KUKA KRL program: EPS_2_251349_MH91A_A_20250929014705.src

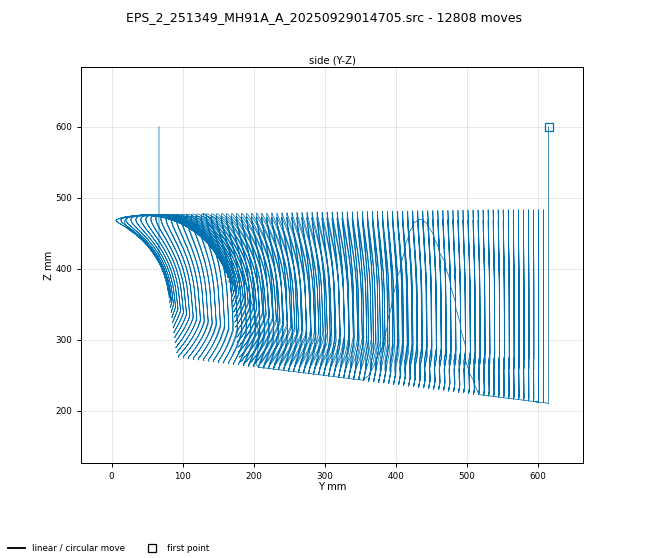
[picture p0: tool path of EPS_2_251349_MH91A_A_20250929014705.src, 12808 of 12810 moves have a stored position in this frame; points joined in program order, loops and branches not executed]
&ACCESS RVP
&REL 4
&COMMENT QRS 19112012
&PARAM EDITMASK = *
DEF PART()
EXT BAS (BAS_COMMAND :IN,REAL :IN )
INT I
BAS (#INITMOV,0 )

;KUKA QRS Post kuka4.cps  Date:22-06-2017 !

File_ID=2865

QRS_PRE_INIT()

;Init var - Until changes are made in qrs_pre_init
Outlet_Square_prg=0
Inlet_1_Square_prg=0
Inlet_2_Square_prg=0
Inlet_3_Square_prg=0
Inlet_4_Square_prg=0
Inlet_5_Square_prg=0

Outlet_1={X 0.000, Y 540.910, Z 382.500, B 0.000, E1 0.000 }
Inlet_1={X 0.000, Y 541.980, Z 367.500, B 0.000, E1 162.000 }
Outlet_1_type=201
Inlet_1_type=201
;QRS#1=Sidecore dimensions
;QRS#2=200-8" PVC SDR 35
;QRS#3=200-8" PVC SDR 35
;QRS#4=
;QRS#5=
;QRS#6=
;QRS#7=
;QRS#8=
;QRS#9=12-08 PSX
;QRS#10=12-08 PSX
;QRS#11=
;QRS#12=
;QRS#13=
;QRS#14=
;QRS#15=
;QRS#16=1220x127x762 2,5'
;QRS#17=EPS Height
;QRS#18=483
;QRS#19=*
;QRS#20= UPDATED VERSION 22-06-2017
;QRS#21=*
Outlet_Square=0100
Inlet_1_Square=0100
Inlet_2_Square=0
Inlet_3_Square=0
Inlet_4_Square=0
Inlet_5_Square=0
Mill_Square=1
Outlet_Square_Prg=204
Inlet_1_Square_prg=204

QRS_INIT()

$ADVANCE=5

; T1
PTP {E1 173.625,E2 173.625}
PTP {X 0,Y 615.486,A -85,B 0,C 180,E1 173.625,E2 173.625,E3 0,E4 0,E5 0,E6 0}
QRS_SPEED_INIT()
LIN {X 0,Y 615.486,Z 600,A -85,B 0,C 180,E1 173.625,E2 173.625,E3 0,E4 0,E5 0,E6 0} C_VEL
LIN {X 0,Y 615.486,Z 220.377,A -85,B 0,C 180,E1 173.625,E2 173.625} C_VEL
LIN {X 0,Y 615.486,Z 212.197,A -85,B 0,C 180,E1 173.625,E2 173.625} C_VEL
LIN {X 0,Y 615.466,Z 210.197,A -85,B 0,C 180,E1 173.439,E2 173.439} C_VEL
LIN {X 0,Y 615.443,Z 210.191,A -85,B 0,C 180,E1 170.804,E2 170.804} C_VEL
LIN {X 0,Y 615.481,Z 210.185,A -85,B 0,C 180,E1 168.143,E2 168.143} C_VEL
LIN {X 0,Y 615.489,Z 210.202,A -85,B 0,C 180,E1 165.455,E2 165.455} C_VEL
LIN {X 0,Y 615.443,Z 210.194,A -85,B 0,C 180,E1 162.732,E2 162.732} C_VEL
LIN {X 0,Y 615.445,Z 210.194,A -85,B 0,C 180,E1 160.665,E2 160.665} C_VEL
LIN {X 0,Y 615.444,Z 210.193,A -85,B 0,C 180,E1 158.571,E2 158.571} C_VEL
LIN {X 0,Y 615.452,Z 210.188,A -85,B 0,C 180,E1 155.999,E2 155.999} C_VEL
LIN {X 0,Y 615.482,Z 210.186,A -85,B 0,C 180,E1 153.56,E2 153.56} C_VEL
LIN {X 0,Y 615.461,Z 210.197,A -85,B 0,C 180,E1 150.597,E2 150.597} C_VEL
LIN {X 0,Y 615.446,Z 210.195,A -85,B 0,C 180,E1 148.317,E2 148.317} C_VEL
LIN {X 0,Y 615.438,Z 210.193,A -85,B 0,C 180,E1 145.98,E2 145.98} C_VEL
LIN {X 0,Y 615.487,Z 210.188,A -85,B 0,C 180,E1 143.064,E2 143.064} C_VEL
LIN {X 0,Y 615.463,Z 210.197,A -85,B 0,C 180,E1 140.254,E2 140.254} C_VEL
LIN {X 0,Y 615.436,Z 210.193,A -85,B 0,C 180,E1 137.649,E2 137.649} C_VEL
LIN {X 0,Y 615.459,Z 210.188,A -85,B 0,C 180,E1 135.071,E2 135.071} C_VEL
LIN {X 0,Y 615.476,Z 210.199,A -85,B 0,C 180,E1 132.086,E2 132.086} C_VEL
LIN {X 0,Y 615.45,Z 210.197,A -85,B 0,C 180,E1 129.753,E2 129.753} C_VEL
LIN {X 0,Y 615.496,Z 210.293,A -85,B 0,C 180,E1 128.068,E2 128.068} C_VEL
LIN {X 0,Y 615.498,Z 215.243,A -85,B 0,C 180,E1 127.241,E2 127.241} C_VEL
LIN {X 0,Y 615.482,Z 234.736,A -85,B 0,C 180,E1 124.194,E2 124.194} C_VEL
LIN {X 0,Y 615.483,Z 252.922,A -85,B 0,C 180,E1 121.388,E2 121.388} C_VEL
LIN {X 0,Y 615.458,Z 256.698,A -85,B 0,C 180,E1 120.85,E2 120.85} C_VEL
LIN {X 0,Y 615.458,Z 257.958,A -85,B 0,C 180,E1 120.802,E2 120.802} C_VEL
LIN {X 0,Y 615.498,Z 364.551,A -85,B 0,C 180,E1 119.531,E2 119.531} C_VEL
LIN {X 0,Y 615.497,Z 378.331,A -85,B 0,C 180,E1 119.218,E2 119.218} C_VEL
LIN {X 0,Y 615.497,Z 390.792,A -85,B 0,C 180,E1 118.798,E2 118.798} C_VEL
LIN {X 0,Y 615.495,Z 402.578,A -85,B 0,C 180,E1 118.257,E2 118.257} C_VEL
LIN {X 0,Y 615.491,Z 414.616,A -85,B 0,C 180,E1 117.545,E2 117.545} C_VEL
LIN {X 0,Y 615.499,Z 425.233,A -85,B 0,C 180,E1 116.751,E2 116.751} C_VEL
LIN {X 0,Y 615.497,Z 434.39,A -85,B 0,C 180,E1 115.897,E2 115.897} C_VEL
LIN {X 0,Y 615.497,Z 442.433,A -85,B 0,C 180,E1 114.991,E2 114.991} C_VEL
LIN {X 0,Y 615.495,Z 449.385,A -85,B 0,C 180,E1 114.023,E2 114.023} C_VEL
LIN {X 0,Y 615.495,Z 454.185,A -85,B 0,C 180,E1 113.2,E2 113.2} C_VEL
LIN {X 0,Y 615.498,Z 459.174,A -85,B 0,C 180,E1 112.136,E2 112.136} C_VEL
LIN {X 0,Y 615.495,Z 462.866,A -85,B 0,C 180,E1 111.081,E2 111.081} C_VEL
LIN {X 0,Y 615.495,Z 465.411,A -85,B 0,C 180,E1 110.033,E2 110.033} C_VEL
LIN {X 0,Y 615.496,Z 466.492,A -85,B 0,C 180,E1 109.338,E2 109.338} C_VEL
LIN {X 0,Y 615.494,Z 467.164,A -85,B 0,C 180,E1 108.624,E2 108.624} C_VEL
LIN {X 0,Y 615.498,Z 467.388,A -85,B 0,C 180,E1 107.957,E2 107.957} C_VEL
LIN {X 0,Y 615.494,Z 467.152,A -85,B 0,C 180,E1 107.27,E2 107.27} C_VEL
LIN {X 0,Y 615.496,Z 466.353,A -85,B 0,C 180,E1 106.453,E2 106.453} C_VEL
LIN {X 0,Y 615.496,Z 463.937,A -85,B 0,C 180,E1 105.226,E2 105.226} C_VEL
LIN {X 0,Y 615.496,Z 459.888,A -85,B 0,C 180,E1 103.959,E2 103.959} C_VEL
LIN {X 0,Y 615.496,Z 455.011,A -85,B 0,C 180,E1 102.865,E2 102.865} C_VEL
LIN {X 0,Y 615.5,Z 448.085,A -85,B 0,C 180,E1 101.694,E2 101.694} C_VEL
LIN {X 0,Y 615.498,Z 440.842,A -85,B 0,C 180,E1 100.724,E2 100.724} C_VEL
LIN {X 0,Y 615.497,Z 434.547,A -85,B 0,C 180,E1 100.028,E2 100.028} C_VEL
LIN {X 0,Y 615.499,Z 425.695,A -85,B 0,C 180,E1 99.199,E2 99.199} C_VEL
LIN {X 0,Y 615.487,Z 415.964,A -85,B 0,C 180,E1 98.454,E2 98.454} C_VEL
LIN {X 0,Y 615.471,Z 405.228,A -85,B 0,C 180,E1 97.793,E2 97.793} C_VEL
LIN {X 0,Y 615.497,Z 393.247,A -85,B 0,C 180,E1 97.216,E2 97.216} C_VEL
LIN {X 0,Y 615.499,Z 381.306,A -85,B 0,C 180,E1 96.78,E2 96.78} C_VEL
LIN {X 0,Y 615.498,Z 368.629,A -85,B 0,C 180,E1 96.454,E2 96.454} C_VEL
LIN {X 0,Y 615.499,Z 353.252,A -85,B 0,C 180,E1 96.228,E2 96.228} C_VEL
LIN {X 0,Y 615.488,Z 257.435,A -85,B 0,C 180,E1 95.098,E2 95.098} C_VEL
LIN {X 0,Y 615.488,Z 256.065,A -85,B 0,C 180,E1 94.995,E2 94.995} C_VEL
LIN {X 0,Y 615.46,Z 238.445,A -85,B 0,C 180,E1 92.291,E2 92.291} C_VEL
LIN {X 0,Y 615.429,Z 222.697,A -85,B 0,C 180,E1 89.837,E2 89.837} C_VEL
LIN {X 0,Y 615.494,Z 210.317,A -85,B 0,C 180,E1 87.853,E2 87.853} C_VEL
LIN {X 0,Y 615.483,Z 210.193,A -85,B 0,C 180,E1 85.416,E2 85.416} C_VEL
LIN {X 0,Y 615.486,Z 210.181,A -85,B 0,C 180,E1 82.785,E2 82.785} C_VEL
LIN {X 0,Y 615.469,Z 210.187,A -85,B 0,C 180,E1 80.138,E2 80.138} C_VEL
LIN {X 0,Y 615.492,Z 210.199,A -85,B 0,C 180,E1 77.47,E2 77.47} C_VEL
LIN {X 0,Y 615.481,Z 210.187,A -85,B 0,C 180,E1 74.774,E2 74.774} C_VEL
LIN {X 0,Y 615.477,Z 210.183,A -85,B 0,C 180,E1 72.043,E2 72.043} C_VEL
LIN {X 0,Y 615.481,Z 210.196,A -85,B 0,C 180,E1 69.269,E2 69.269} C_VEL
LIN {X 0,Y 615.482,Z 210.187,A -85,B 0,C 180,E1 66.444,E2 66.444} C_VEL
LIN {X 0,Y 615.479,Z 210.186,A -85,B 0,C 180,E1 64.284,E2 64.284} C_VEL
LIN {X 0,Y 615.471,Z 210.185,A -85,B 0,C 180,E1 61.541,E2 61.541} C_VEL
LIN {X 0,Y 615.477,Z 210.195,A -85,B 0,C 180,E1 58.906,E2 58.906} C_VEL
LIN {X 0,Y 615.492,Z 210.197,A -85,B 0,C 180,E1 56.456,E2 56.456} C_VEL
LIN {X 0,Y 615.483,Z 210.181,A -85,B 0,C 180,E1 53.575,E2 53.575} C_VEL
LIN {X 0,Y 615.467,Z 210.188,A -85,B 0,C 180,E1 50.932,E2 50.932} C_VEL
LIN {X 0,Y 615.476,Z 210.195,A -85,B 0,C 180,E1 48.526,E2 48.526} C_VEL
LIN {X 0,Y 615.484,Z 210.193,A -85,B 0,C 180,E1 45.851,E2 45.851} C_VEL
LIN {X 0,Y 615.483,Z 210.181,A -85,B 0,C 180,E1 43.048,E2 43.048} C_VEL
LIN {X 0,Y 615.468,Z 210.187,A -85,B 0,C 180,E1 40.602,E2 40.602} C_VEL
LIN {X 0,Y 615.477,Z 210.198,A -85,B 0,C 180,E1 38.011,E2 38.011} C_VEL
LIN {X 0,Y 615.491,Z 210.197,A -85,B 0,C 180,E1 35.61,E2 35.61} C_VEL
LIN {X 0,Y 615.482,Z 210.189,A -85,B 0,C 180,E1 33.231,E2 33.231} C_VEL
LIN {X 0,Y 615.484,Z 210.184,A -85,B 0,C 180,E1 30.915,E2 30.915} C_VEL
LIN {X 0,Y 615.482,Z 210.181,A -85,B 0,C 180,E1 28.45,E2 28.45} C_VEL
LIN {X 0,Y 615.478,Z 210.196,A -85,B 0,C 180,E1 25.568,E2 25.568} C_VEL
LIN {X 0,Y 615.482,Z 210.19,A -85,B 0,C 180,E1 22.84,E2 22.84} C_VEL
LIN {X 0,Y 615.477,Z 210.182,A -85,B 0,C 180,E1 20.029,E2 20.029} C_VEL
LIN {X 0,Y 615.473,Z 210.196,A -85,B 0,C 180,E1 17.267,E2 17.267} C_VEL
LIN {X 0,Y 615.483,Z 210.191,A -85,B 0,C 180,E1 14.545,E2 14.545} C_VEL
LIN {X 0,Y 615.485,Z 210.181,A -85,B 0,C 180,E1 11.857,E2 11.857} C_VEL
LIN {X 0,Y 615.466,Z 210.191,A -85,B 0,C 180,E1 9.196,E2 9.196} C_VEL
LIN {X 0,Y 615.489,Z 210.201,A -85,B 0,C 180,E1 6.553,E2 6.553} C_VEL
LIN {X 0,Y 615.485,Z 210.185,A -85,B 0,C 180,E1 3.925,E2 3.925} C_VEL
LIN {X 0,Y 615.477,Z 210.182,A -85,B 0,C 180,E1 1.306,E2 1.306} C_VEL
LIN {X 0,Y 615.468,Z 210.192,A -85,B 0,C 180,E1 -1.312,E2 -1.312} C_VEL
LIN {X 0,Y 615.488,Z 210.199,A -85,B 0,C 180,E1 -3.931,E2 -3.931} C_VEL
LIN {X 0,Y 615.484,Z 210.184,A -85,B 0,C 180,E1 -6.58,E2 -6.58} C_VEL
LIN {X 0,Y 615.471,Z 210.184,A -85,B 0,C 180,E1 -9.202,E2 -9.202} C_VEL
LIN {X 0,Y 615.474,Z 210.195,A -85,B 0,C 180,E1 -11.863,E2 -11.863} C_VEL
LIN {X 0,Y 615.484,Z 210.192,A -85,B 0,C 180,E1 -14.551,E2 -14.551} C_VEL
LIN {X 0,Y 615.487,Z 210.18,A -85,B 0,C 180,E1 -17.273,E2 -17.273} C_VEL
LIN {X 0,Y 615.465,Z 210.192,A -85,B 0,C 180,E1 -20.036,E2 -20.036} C_VEL
LIN {X 0,Y 615.486,Z 210.193,A -85,B 0,C 180,E1 -22.847,E2 -22.847} C_VEL
LIN {X 0,Y 615.479,Z 210.182,A -85,B 0,C 180,E1 -25.718,E2 -25.718} C_VEL
LIN {X 0,Y 615.47,Z 210.194,A -85,B 0,C 180,E1 -28.448,E2 -28.448} C_VEL
LIN {X 0,Y 615.483,Z 210.197,A -85,B 0,C 180,E1 -31.086,E2 -31.086} C_VEL
LIN {X 0,Y 615.478,Z 210.182,A -85,B 0,C 180,E1 -34.024,E2 -34.024} C_VEL
LIN {X 0,Y 615.463,Z 210.188,A -85,B 0,C 180,E1 -36.428,E2 -36.428} C_VEL
LIN {X 0,Y 615.483,Z 210.197,A -85,B 0,C 180,E1 -39.062,E2 -39.062} C_VEL
LIN {X 0,Y 615.49,Z 210.196,A -85,B 0,C 180,E1 -41.475,E2 -41.475} C_VEL
LIN {X 0,Y 615.495,Z 210.18,A -85,B 0,C 180,E1 -44.15,E2 -44.15} C_VEL
LIN {X 0,Y 615.463,Z 210.19,A -85,B 0,C 180,E1 -46.956,E2 -46.956} C_VEL
LIN {X 0,Y 615.477,Z 210.196,A -85,B 0,C 180,E1 -49.393,E2 -49.393} C_VEL
LIN {X 0,Y 615.486,Z 210.193,A -85,B 0,C 180,E1 -51.99,E2 -51.99} C_VEL
LIN {X 0,Y 615.487,Z 210.185,A -85,B 0,C 180,E1 -54.385,E2 -54.385} C_VEL
LIN {X 0,Y 615.487,Z 210.181,A -85,B 0,C 180,E1 -56.764,E2 -56.764} C_VEL
LIN {X 0,Y 615.474,Z 210.183,A -85,B 0,C 180,E1 -59.08,E2 -59.08} C_VEL
LIN {X 0,Y 615.463,Z 210.19,A -85,B 0,C 180,E1 -61.555,E2 -61.555} C_VEL
LIN {X 0,Y 615.496,Z 210.198,A -85,B 0,C 180,E1 -64.285,E2 -64.285} C_VEL
LIN {X 0,Y 615.484,Z 210.181,A -85,B 0,C 180,E1 -67.156,E2 -67.156} C_VEL
LIN {X 0,Y 615.492,Z 210.44,A -85,B 0,C 180,E1 -68.481,E2 -68.481} C_VEL
LIN {X 0,Y 615.494,Z 228.962,A -85,B 0,C 180,E1 -71.182,E2 -71.182} C_VEL
LIN {X 0,Y 615.488,Z 249.426,A -85,B 0,C 180,E1 -74.095,E2 -74.095} C_VEL
LIN {X 0,Y 615.473,Z 268.666,A -85,B 0,C 180,E1 -76.799,E2 -76.799} C_VEL
LIN {X 0,Y 615.487,Z 271.254,A -85,B 0,C 180,E1 -77.114,E2 -77.114} C_VEL
LIN {X 0,Y 615.491,Z 280.067,A -85,B 0,C 180,E1 -77.24,E2 -77.24} C_VEL
LIN {X 0,Y 615.498,Z 378.843,A -85,B 0,C 180,E1 -78.411,E2 -78.411} C_VEL
LIN {X 0,Y 615.498,Z 391.352,A -85,B 0,C 180,E1 -78.682,E2 -78.682} C_VEL
LIN {X 0,Y 615.496,Z 404.516,A -85,B 0,C 180,E1 -79.109,E2 -79.109} C_VEL
LIN {X 0,Y 615.491,Z 416.482,A -85,B 0,C 180,E1 -79.64,E2 -79.64} C_VEL
LIN {X 0,Y 615.48,Z 428,A -85,B 0,C 180,E1 -80.304,E2 -80.304} C_VEL
LIN {X 0,Y 615.499,Z 438.344,A -85,B 0,C 180,E1 -81.05,E2 -81.05} C_VEL
LIN {X 0,Y 615.498,Z 446.694,A -85,B 0,C 180,E1 -81.794,E2 -81.794} C_VEL
LIN {X 0,Y 615.498,Z 454.608,A -85,B 0,C 180,E1 -82.62,E2 -82.62} C_VEL
LIN {X 0,Y 615.49,Z 462.206,A -85,B 0,C 180,E1 -83.608,E2 -83.608} C_VEL
LIN {X 0,Y 615.498,Z 469.206,A -85,B 0,C 180,E1 -84.759,E2 -84.759} C_VEL
LIN {X 0,Y 615.493,Z 473.852,A -85,B 0,C 180,E1 -85.744,E2 -85.744} C_VEL
LIN {X 0,Y 615.494,Z 477.399,A -85,B 0,C 180,E1 -86.727,E2 -86.727} C_VEL
LIN {X 0,Y 615.497,Z 479.233,A -85,B 0,C 180,E1 -87.382,E2 -87.382} C_VEL
LIN {X 0,Y 615.497,Z 480.609,A -85,B 0,C 180,E1 -88.037,E2 -88.037} C_VEL
LIN {X 0,Y 615.496,Z 482.174,A -85,B 0,C 180,E1 -89.346,E2 -89.346} C_VEL
LIN {X 0,Y 615.494,Z 482.389,A -85,B 0,C 180,E1 -90,E2 -90} C_VEL
LIN {X 0,Y 615.495,Z 481.58,A -85,B 0,C 180,E1 -91.309,E2 -91.309} C_VEL
LIN {X 0,Y 615.497,Z 480.608,A -85,B 0,C 180,E1 -91.963,E2 -91.963} C_VEL
LIN {X 0,Y 615.497,Z 479.232,A -85,B 0,C 180,E1 -92.618,E2 -92.618} C_VEL
LIN {X 0,Y 615.496,Z 476.349,A -85,B 0,C 180,E1 -93.601,E2 -93.601} C_VEL
LIN {X 0,Y 615.498,Z 472.441,A -85,B 0,C 180,E1 -94.585,E2 -94.585} C_VEL
LIN {X 0,Y 615.499,Z 467.404,A -85,B 0,C 180,E1 -95.57,E2 -95.57} C_VEL
LIN {X 0,Y 615.489,Z 460.919,A -85,B 0,C 180,E1 -96.577,E2 -96.577} C_VEL
LIN {X 0,Y 615.497,Z 453.131,A -85,B 0,C 180,E1 -97.546,E2 -97.546} C_VEL
LIN {X 0,Y 615.498,Z 443.255,A -85,B 0,C 180,E1 -98.537,E2 -98.537} C_VEL
LIN {X 0,Y 615.495,Z 432.863,A -85,B 0,C 180,E1 -99.365,E2 -99.365} C_VEL
LIN {X 0,Y 615.475,Z 422.574,A -85,B 0,C 180,E1 -100.029,E2 -100.029} C_VEL
LIN {X 0,Y 615.497,Z 411.095,A -85,B 0,C 180,E1 -100.618,E2 -100.618} C_VEL
LIN {X 0,Y 615.499,Z 399.268,A -85,B 0,C 180,E1 -101.08,E2 -101.08} C_VEL
LIN {X 0,Y 615.498,Z 386.231,A -85,B 0,C 180,E1 -101.443,E2 -101.443} C_VEL
LIN {X 0,Y 615.499,Z 372.923,A -85,B 0,C 180,E1 -101.673,E2 -101.673} C_VEL
LIN {X 0,Y 615.487,Z 271.727,A -85,B 0,C 180,E1 -102.866,E2 -102.866} C_VEL
LIN {X 0,Y 615.485,Z 270.517,A -85,B 0,C 180,E1 -102.95,E2 -102.95} C_VEL
LIN {X 0,Y 615.482,Z 250.626,A -85,B 0,C 180,E1 -105.735,E2 -105.735} C_VEL
LIN {X 0,Y 615.491,Z 231.585,A -85,B 0,C 180,E1 -108.443,E2 -108.443} C_VEL
LIN {X 0,Y 615.492,Z 212.09,A -85,B 0,C 180,E1 -111.256,E2 -111.256} C_VEL
LIN {X 0,Y 615.49,Z 210.313,A -85,B 0,C 180,E1 -111.564,E2 -111.564} C_VEL
LIN {X 0,Y 615.462,Z 210.19,A -85,B 0,C 180,E1 -114.273,E2 -114.273} C_VEL
LIN {X 0,Y 615.497,Z 210.179,A -85,B 0,C 180,E1 -117.045,E2 -117.045} C_VEL
LIN {X 0,Y 615.493,Z 210.197,A -85,B 0,C 180,E1 -119.794,E2 -119.794} C_VEL
LIN {X 0,Y 615.463,Z 210.192,A -85,B 0,C 180,E1 -122.459,E2 -122.459} C_VEL
LIN {X 0,Y 615.46,Z 210.188,A -85,B 0,C 180,E1 -124.817,E2 -124.817} C_VEL
LIN {X 0,Y 615.478,Z 210.182,A -85,B 0,C 180,E1 -127.243,E2 -127.243} C_VEL
LIN {X 0,Y 615.49,Z 210.195,A -85,B 0,C 180,E1 -130.088,E2 -130.088} C_VEL
LIN {X 0,Y 615.499,Z 210.2,A -85,B 0,C 180,E1 -132.352,E2 -132.352} C_VEL
LIN {X 0,Y 615.455,Z 210.191,A -85,B 0,C 180,E1 -135.072,E2 -135.072} C_VEL
LIN {X 0,Y 615.497,Z 210.181,A -85,B 0,C 180,E1 -137.919,E2 -137.919} C_VEL
LIN {X 0,Y 615.487,Z 210.189,A -85,B 0,C 180,E1 -140.248,E2 -140.248} C_VEL
LIN {X 0,Y 615.467,Z 210.195,A -85,B 0,C 180,E1 -143.066,E2 -143.066} C_VEL
LIN {X 0,Y 615.458,Z 210.193,A -85,B 0,C 180,E1 -145.303,E2 -145.303} C_VEL
LIN {X 0,Y 615.456,Z 210.189,A -85,B 0,C 180,E1 -147.674,E2 -147.674} C_VEL
LIN {X 0,Y 615.482,Z 210.183,A -85,B 0,C 180,E1 -150.206,E2 -150.206} C_VEL
LIN {X 0,Y 615.493,Z 210.196,A -85,B 0,C 180,E1 -152.954,E2 -152.954} C_VEL
LIN {X 0,Y 615.452,Z 210.193,A -85,B 0,C 180,E1 -155.724,E2 -155.724} C_VEL
LIN {X 0,Y 615.453,Z 210.192,A -85,B 0,C 180,E1 -157.86,E2 -157.86} C_VEL
LIN {X 0,Y 615.45,Z 210.192,A -85,B 0,C 180,E1 -159.964,E2 -159.964} C_VEL
LIN {X 0,Y 615.452,Z 210.191,A -85,B 0,C 180,E1 -162.04,E2 -162.04} C_VEL
LIN {X 0,Y 615.483,Z 210.183,A -85,B 0,C 180,E1 -164.772,E2 -164.772} C_VEL
LIN {X 0,Y 615.489,Z 210.197,A -85,B 0,C 180,E1 -167.467,E2 -167.467} C_VEL
LIN {X 0,Y 615.457,Z 210.194,A -85,B 0,C 180,E1 -170.135,E2 -170.135} C_VEL
LIN {X 0,Y 615.457,Z 210.187,A -85,B 0,C 180,E1 -172.781,E2 -172.781} C_VEL
LIN {X 0,Y 615.495,Z 210.185,A -85,B 0,C 180,E1 -175.413,E2 -175.413} C_VEL
LIN {X 0,Y 615.492,Z 210.199,A -85,B 0,C 180,E1 -178.034,E2 -178.034} C_VEL
LIN {X 0,Y 615.449,Z 210.193,A -85,B 0,C 180,E1 -180.651,E2 -180.651} C_VEL
LIN {X 0,Y 615.46,Z 210.187,A -85,B 0,C 180,E1 -183.27,E2 -183.27} C_VEL
LIN {X 0,Y 615.494,Z 210.188,A -85,B 0,C 180,E1 -185.895,E2 -185.895} C_VEL
LIN {X 0,Y 615.466,Z 210.197,A -85,B 0,C 180,E1 -186.561,E2 -186.561} C_VEL
LIN {X 0,Y 614.775,Z 210.337,A -85,B 0,C 180,E1 -187.107,E2 -187.107} C_VEL
LIN {X 0,Y 611.924,Z 210.759,A -85,B 0,C 180,E1 -187.993,E2 -187.993} C_VEL
LIN {X 0,Y 609.535,Z 211.065,A -85,B 0,C 180,E1 -188.706,E2 -188.706} C_VEL
LIN {X 0,Y 608.516,Z 211.18,A -85,B 0,C 180,E1 -189.256,E2 -189.256} C_VEL
LIN {X 0,Y 608.436,Z 211.188,A -85,B 0,C 180,E1 -189.442,E2 -189.442} C_VEL
LIN {X 0,Y 608.458,Z 211.189,A -85,B 0,C 180,E1 -191.996,E2 -191.996} C_VEL
LIN {X 0,Y 608.466,Z 211.193,A -85,B 0,C 180,E1 -194.717,E2 -194.717} C_VEL
LIN {X 0,Y 608.419,Z 211.191,A -85,B 0,C 180,E1 -197.474,E2 -197.474} C_VEL
LIN {X 0,Y 608.421,Z 211.19,A -85,B 0,C 180,E1 -199.568,E2 -199.568} C_VEL
LIN {X 0,Y 608.436,Z 211.188,A -85,B 0,C 180,E1 -201.688,E2 -201.688} C_VEL
LIN {X 0,Y 608.447,Z 211.192,A -85,B 0,C 180,E1 -204.567,E2 -204.567} C_VEL
LIN {X 0,Y 608.425,Z 211.193,A -85,B 0,C 180,E1 -207.514,E2 -207.514} C_VEL
LIN {X 0,Y 608.426,Z 211.19,A -85,B 0,C 180,E1 -209.965,E2 -209.965} C_VEL
LIN {X 0,Y 608.437,Z 211.189,A -85,B 0,C 180,E1 -212.519,E2 -212.519} C_VEL
LIN {X 0,Y 608.432,Z 211.2,A -85,B 0,C 180,E1 -215.273,E2 -215.273} C_VEL
LIN {X 0,Y 608.441,Z 211.193,A -85,B 0,C 180,E1 -217.743,E2 -217.743} C_VEL
LIN {X 0,Y 608.409,Z 211.192,A -85,B 0,C 180,E1 -220.324,E2 -220.324} C_VEL
LIN {X 0,Y 608.436,Z 211.19,A -85,B 0,C 180,E1 -222.955,E2 -222.955} C_VEL
LIN {X 0,Y 608.441,Z 211.199,A -85,B 0,C 180,E1 -225.731,E2 -225.731} C_VEL
LIN {X 0,Y 608.453,Z 211.194,A -85,B 0,C 180,E1 -227.938,E2 -227.938} C_VEL
LIN {X 0,Y 608.433,Z 211.19,A -85,B 0,C 180,E1 -230.699,E2 -230.699} C_VEL
LIN {X 0,Y 608.503,Z 211.414,A -85,B 0,C 180,E1 -231.896,E2 -231.896} C_VEL
LIN {X 0,Y 608.479,Z 227.922,A -85,B 0,C 180,E1 -234.529,E2 -234.529} C_VEL
LIN {X 0,Y 608.48,Z 244.489,A -85,B 0,C 180,E1 -237.122,E2 -237.122} C_VEL
LIN {X 0,Y 608.457,Z 256.895,A -85,B 0,C 180,E1 -239.009,E2 -239.009} C_VEL
LIN {X 0,Y 608.559,Z 259.904,A -85,B 0,C 180,E1 -239.075,E2 -239.075} C_VEL
LIN {X 0,Y 608.55,Z 364.504,A -85,B 0,C 180,E1 -240.332,E2 -240.332} C_VEL
LIN {X 0,Y 608.543,Z 377.632,A -85,B 0,C 180,E1 -240.629,E2 -240.629} C_VEL
LIN {X 0,Y 608.532,Z 389.978,A -85,B 0,C 180,E1 -241.041,E2 -241.041} C_VEL
LIN {X 0,Y 608.511,Z 402.259,A -85,B 0,C 180,E1 -241.598,E2 -241.598} C_VEL
LIN {X 0,Y 608.498,Z 414.13,A -85,B 0,C 180,E1 -242.298,E2 -242.298} C_VEL
LIN {X 0,Y 608.487,Z 424.611,A -85,B 0,C 180,E1 -243.072,E2 -243.072} C_VEL
LIN {X 0,Y 608.458,Z 434.253,A -85,B 0,C 180,E1 -243.965,E2 -243.965} C_VEL
LIN {X 0,Y 608.455,Z 442.443,A -85,B 0,C 180,E1 -244.882,E2 -244.882} C_VEL
LIN {X 0,Y 608.454,Z 449.372,A -85,B 0,C 180,E1 -245.839,E2 -245.839} C_VEL
LIN {X 0,Y 608.436,Z 455.39,A -85,B 0,C 180,E1 -246.875,E2 -246.875} C_VEL
LIN {X 0,Y 608.452,Z 460.23,A -85,B 0,C 180,E1 -247.951,E2 -247.951} C_VEL
LIN {X 0,Y 608.438,Z 463.798,A -85,B 0,C 180,E1 -249.018,E2 -249.018} C_VEL
LIN {X 0,Y 608.434,Z 465.533,A -85,B 0,C 180,E1 -249.725,E2 -249.725} C_VEL
LIN {X 0,Y 608.436,Z 466.815,A -85,B 0,C 180,E1 -250.429,E2 -250.429} C_VEL
LIN {X 0,Y 608.437,Z 467.708,A -85,B 0,C 180,E1 -251.276,E2 -251.276} C_VEL
LIN {X 0,Y 608.437,Z 467.894,A -85,B 0,C 180,E1 -252.523,E2 -252.523} C_VEL
LIN {X 0,Y 608.424,Z 467.07,A -85,B 0,C 180,E1 -253.466,E2 -253.466} C_VEL
LIN {X 0,Y 608.42,Z 465.042,A -85,B 0,C 180,E1 -254.593,E2 -254.593} C_VEL
LIN {X 0,Y 608.441,Z 462.112,A -85,B 0,C 180,E1 -255.62,E2 -255.62} C_VEL
LIN {X 0,Y 608.442,Z 458.121,A -85,B 0,C 180,E1 -256.643,E2 -256.643} C_VEL
LIN {X 0,Y 608.437,Z 451.97,A -85,B 0,C 180,E1 -257.83,E2 -257.83} C_VEL
LIN {X 0,Y 608.445,Z 444.669,A -85,B 0,C 180,E1 -258.921,E2 -258.921} C_VEL
LIN {X 0,Y 608.477,Z 436.901,A -85,B 0,C 180,E1 -259.855,E2 -259.855} C_VEL
LIN {X 0,Y 608.467,Z 426.444,A -85,B 0,C 180,E1 -260.862,E2 -260.862} C_VEL
LIN {X 0,Y 608.471,Z 415.564,A -85,B 0,C 180,E1 -261.699,E2 -261.699} C_VEL
LIN {X 0,Y 608.492,Z 404.602,A -85,B 0,C 180,E1 -262.367,E2 -262.367} C_VEL
LIN {X 0,Y 608.542,Z 391.798,A -85,B 0,C 180,E1 -262.976,E2 -262.976} C_VEL
LIN {X 0,Y 608.532,Z 379.509,A -85,B 0,C 180,E1 -263.41,E2 -263.41} C_VEL
LIN {X 0,Y 608.565,Z 366.436,A -85,B 0,C 180,E1 -263.722,E2 -263.722} C_VEL
LIN {X 0,Y 608.55,Z 346.3,A -85,B 0,C 180,E1 -263.992,E2 -263.992} C_VEL
LIN {X 0,Y 608.537,Z 257.452,A -85,B 0,C 180,E1 -265.052,E2 -265.052} C_VEL
LIN {X 0,Y 608.463,Z 256.535,A -85,B 0,C 180,E1 -265.113,E2 -265.113} C_VEL
LIN {X 0,Y 608.458,Z 238.843,A -85,B 0,C 180,E1 -267.848,E2 -267.848} C_VEL
LIN {X 0,Y 608.447,Z 223.051,A -85,B 0,C 180,E1 -270.331,E2 -270.331} C_VEL
LIN {X 0,Y 608.5,Z 211.284,A -85,B 0,C 180,E1 -272.234,E2 -272.234} C_VEL
LIN {X 0,Y 608.485,Z 211.182,A -85,B 0,C 180,E1 -275.301,E2 -275.301} C_VEL
LIN {X 0,Y 608.456,Z 211.189,A -85,B 0,C 180,E1 -277.967,E2 -277.967} C_VEL
LIN {X 0,Y 608.462,Z 211.195,A -85,B 0,C 180,E1 -280.65,E2 -280.65} C_VEL
LIN {X 0,Y 608.454,Z 211.187,A -85,B 0,C 180,E1 -283.356,E2 -283.356} C_VEL
LIN {X 0,Y 608.467,Z 211.186,A -85,B 0,C 180,E1 -286.093,E2 -286.093} C_VEL
LIN {X 0,Y 608.453,Z 211.198,A -85,B 0,C 180,E1 -288.869,E2 -288.869} C_VEL
LIN {X 0,Y 608.457,Z 211.186,A -85,B 0,C 180,E1 -291.692,E2 -291.692} C_VEL
LIN {X 0,Y 608.44,Z 211.19,A -85,B 0,C 180,E1 -294.571,E2 -294.571} C_VEL
LIN {X 0,Y 608.469,Z 211.195,A -85,B 0,C 180,E1 -297.217,E2 -297.217} C_VEL
LIN {X 0,Y 608.484,Z 211.183,A -85,B 0,C 180,E1 -299.985,E2 -299.985} C_VEL
LIN {X 0,Y 608.447,Z 211.189,A -85,B 0,C 180,E1 -302.88,E2 -302.88} C_VEL
LIN {X 0,Y 608.466,Z 211.192,A -85,B 0,C 180,E1 -305.276,E2 -305.276} C_VEL
LIN {X 0,Y 608.455,Z 211.188,A -85,B 0,C 180,E1 -308.247,E2 -308.247} C_VEL
LIN {X 0,Y 608.472,Z 211.185,A -85,B 0,C 180,E1 -310.339,E2 -310.339} C_VEL
LIN {X 0,Y 608.454,Z 211.189,A -85,B 0,C 180,E1 -313.314,E2 -313.314} C_VEL
LIN {X 0,Y 608.47,Z 211.192,A -85,B 0,C 180,E1 -316.137,E2 -316.137} C_VEL
LIN {X 0,Y 608.455,Z 211.186,A -85,B 0,C 180,E1 -318.83,E2 -318.83} C_VEL
LIN {X 0,Y 608.462,Z 211.185,A -85,B 0,C 180,E1 -321.417,E2 -321.417} C_VEL
LIN {X 0,Y 608.456,Z 211.192,A -85,B 0,C 180,E1 -323.953,E2 -323.953} C_VEL
LIN {X 0,Y 608.461,Z 211.197,A -85,B 0,C 180,E1 -326.334,E2 -326.334} C_VEL
LIN {X 0,Y 608.46,Z 211.191,A -85,B 0,C 180,E1 -328.73,E2 -328.73} C_VEL
LIN {X 0,Y 608.468,Z 211.184,A -85,B 0,C 180,E1 -331.38,E2 -331.38} C_VEL
LIN {X 0,Y 608.436,Z 211.189,A -85,B 0,C 180,E1 -333.969,E2 -333.969} C_VEL
LIN {X 0,Y 608.451,Z 211.188,A -85,B 0,C 180,E1 -336.159,E2 -336.159} C_VEL
LIN {X 0,Y 608.455,Z 211.189,A -85,B 0,C 180,E1 -338.312,E2 -338.312} C_VEL
LIN {X 0,Y 608.446,Z 211.194,A -85,B 0,C 180,E1 -341.134,E2 -341.134} C_VEL
LIN {X 0,Y 608.455,Z 211.185,A -85,B 0,C 180,E1 -343.91,E2 -343.91} C_VEL
LIN {X 0,Y 608.452,Z 211.189,A -85,B 0,C 180,E1 -346.647,E2 -346.647} C_VEL
LIN {X 0,Y 608.464,Z 211.195,A -85,B 0,C 180,E1 -349.354,E2 -349.354} C_VEL
LIN {X 0,Y 608.477,Z 211.184,A -85,B 0,C 180,E1 -352.036,E2 -352.036} C_VEL
LIN {X 0,Y 608.449,Z 211.187,A -85,B 0,C 180,E1 -354.701,E2 -354.701} C_VEL
LIN {X 0,Y 608.472,Z 211.191,A -85,B 0,C 180,E1 -357.355,E2 -357.355} C_VEL
LIN {X 0,Y 608.474,Z 211.189,A -85,B 0,C 180,E1 -360.003,E2 -360.003} C_VEL
LIN {X 0,Y 608.481,Z 211.183,A -85,B 0,C 180,E1 -362.651,E2 -362.651} C_VEL
LIN {X 0,Y 608.448,Z 211.189,A -85,B 0,C 180,E1 -365.305,E2 -365.305} C_VEL
LIN {X 0,Y 608.476,Z 211.195,A -85,B 0,C 180,E1 -367.97,E2 -367.97} C_VEL
LIN {X 0,Y 608.469,Z 211.184,A -85,B 0,C 180,E1 -370.958,E2 -370.958} C_VEL
LIN {X 0,Y 608.456,Z 211.186,A -85,B 0,C 180,E1 -373.359,E2 -373.359} C_VEL
LIN {X 0,Y 608.451,Z 211.194,A -85,B 0,C 180,E1 -376.096,E2 -376.096} C_VEL
LIN {X 0,Y 608.458,Z 211.189,A -85,B 0,C 180,E1 -378.872,E2 -378.872} C_VEL
LIN {X 0,Y 608.463,Z 211.185,A -85,B 0,C 180,E1 -381.694,E2 -381.694} C_VEL
LIN {X 0,Y 608.445,Z 211.198,A -85,B 0,C 180,E1 -384.573,E2 -384.573} C_VEL
LIN {X 0,Y 608.478,Z 211.187,A -85,B 0,C 180,E1 -387.208,E2 -387.208} C_VEL
LIN {X 0,Y 608.443,Z 211.187,A -85,B 0,C 180,E1 -389.968,E2 -389.968} C_VEL
LIN {X 0,Y 608.45,Z 211.196,A -85,B 0,C 180,E1 -392.882,E2 -392.882} C_VEL
LIN {X 0,Y 608.438,Z 211.196,A -85,B 0,C 180,E1 -395.28,E2 -395.28} C_VEL
LIN {X 0,Y 608.47,Z 211.186,A -85,B 0,C 180,E1 -397.748,E2 -397.748} C_VEL
LIN {X 0,Y 608.447,Z 211.187,A -85,B 0,C 180,E1 -400.329,E2 -400.329} C_VEL
LIN {X 0,Y 608.437,Z 211.192,A -85,B 0,C 180,E1 -402.963,E2 -402.963} C_VEL
LIN {X 0,Y 608.453,Z 211.193,A -85,B 0,C 180,E1 -405.738,E2 -405.738} C_VEL
LIN {X 0,Y 608.452,Z 211.186,A -85,B 0,C 180,E1 -408.66,E2 -408.66} C_VEL
LIN {X 0,Y 608.467,Z 211.196,A -85,B 0,C 180,E1 -411.761,E2 -411.761} C_VEL
LIN {X 0,Y 608.436,Z 211.188,A -85,B 0,C 180,E1 -414.722,E2 -414.722} C_VEL
LIN {X 0,Y 608.452,Z 211.187,A -85,B 0,C 180,E1 -417.121,E2 -417.121} C_VEL
LIN {X 0,Y 608.468,Z 211.196,A -85,B 0,C 180,E1 -420.03,E2 -420.03} C_VEL
LIN {X 0,Y 608.486,Z 211.184,A -85,B 0,C 180,E1 -422.793,E2 -422.793} C_VEL
LIN {X 0,Y 608.445,Z 211.188,A -85,B 0,C 180,E1 -425.429,E2 -425.429} C_VEL
LIN {X 0,Y 608.5,Z 211.351,A -85,B 0,C 180,E1 -428.354,E2 -428.354} C_VEL
LIN {X 0,Y 608.545,Z 226.58,A -85,B 0,C 180,E1 -430.608,E2 -430.608} C_VEL
LIN {X 0,Y 608.505,Z 246.378,A -85,B 0,C 180,E1 -433.461,E2 -433.461} C_VEL
LIN {X 0,Y 608.467,Z 266.398,A -85,B 0,C 180,E1 -436.304,E2 -436.304} C_VEL
LIN {X 0,Y 608.497,Z 271.295,A -85,B 0,C 180,E1 -436.963,E2 -436.963} C_VEL
LIN {X 0,Y 608.587,Z 276.532,A -85,B 0,C 180,E1 -437.05,E2 -437.05} C_VEL
LIN {X 0,Y 608.548,Z 378.962,A -85,B 0,C 180,E1 -438.277,E2 -438.277} C_VEL
LIN {X 0,Y 608.548,Z 392.226,A -85,B 0,C 180,E1 -438.572,E2 -438.572} C_VEL
LIN {X 0,Y 608.544,Z 405.347,A -85,B 0,C 180,E1 -439.01,E2 -439.01} C_VEL
LIN {X 0,Y 608.516,Z 416.64,A -85,B 0,C 180,E1 -439.52,E2 -439.52} C_VEL
LIN {X 0,Y 608.468,Z 428.201,A -85,B 0,C 180,E1 -440.191,E2 -440.191} C_VEL
LIN {X 0,Y 608.485,Z 438.597,A -85,B 0,C 180,E1 -440.946,E2 -440.946} C_VEL
LIN {X 0,Y 608.459,Z 447.005,A -85,B 0,C 180,E1 -441.699,E2 -441.699} C_VEL
LIN {X 0,Y 608.471,Z 454.962,A -85,B 0,C 180,E1 -442.534,E2 -442.534} C_VEL
LIN {X 0,Y 608.436,Z 462.304,A -85,B 0,C 180,E1 -443.487,E2 -443.487} C_VEL
LIN {X 0,Y 608.45,Z 467.867,A -85,B 0,C 180,E1 -444.366,E2 -444.366} C_VEL
LIN {X 0,Y 608.432,Z 472.951,A -85,B 0,C 180,E1 -445.362,E2 -445.362} C_VEL
LIN {X 0,Y 608.449,Z 476.897,A -85,B 0,C 180,E1 -446.358,E2 -446.358} C_VEL
LIN {X 0,Y 608.425,Z 479.81,A -85,B 0,C 180,E1 -447.352,E2 -447.352} C_VEL
LIN {X 0,Y 608.442,Z 481.202,A -85,B 0,C 180,E1 -448.014,E2 -448.014} C_VEL
LIN {X 0,Y 608.439,Z 482.784,A -85,B 0,C 180,E1 -449.338,E2 -449.338} C_VEL
LIN {X 0,Y 608.434,Z 483,A -85,B 0,C 180,E1 -450,E2 -450} C_VEL
LIN {X 0,Y 608.448,Z 482.184,A -85,B 0,C 180,E1 -451.324,E2 -451.324} C_VEL
LIN {X 0,Y 608.442,Z 481.201,A -85,B 0,C 180,E1 -451.986,E2 -451.986} C_VEL
LIN {X 0,Y 608.425,Z 479.809,A -85,B 0,C 180,E1 -452.648,E2 -452.648} C_VEL
LIN {X 0,Y 608.449,Z 476.895,A -85,B 0,C 180,E1 -453.643,E2 -453.643} C_VEL
LIN {X 0,Y 608.432,Z 472.949,A -85,B 0,C 180,E1 -454.638,E2 -454.638} C_VEL
LIN {X 0,Y 608.437,Z 466.875,A -85,B 0,C 180,E1 -455.801,E2 -455.801} C_VEL
LIN {X 0,Y 608.462,Z 460.234,A -85,B 0,C 180,E1 -456.799,E2 -456.799} C_VEL
LIN {X 0,Y 608.456,Z 451.987,A -85,B 0,C 180,E1 -457.8,E2 -457.8} C_VEL
LIN {X 0,Y 608.477,Z 441.596,A -85,B 0,C 180,E1 -458.803,E2 -458.803} C_VEL
LIN {X 0,Y 608.486,Z 430.744,A -85,B 0,C 180,E1 -459.641,E2 -459.641} C_VEL
LIN {X 0,Y 608.489,Z 419.77,A -85,B 0,C 180,E1 -460.313,E2 -460.313} C_VEL
LIN {X 0,Y 608.537,Z 407.791,A -85,B 0,C 180,E1 -460.889,E2 -460.889} C_VEL
LIN {X 0,Y 608.534,Z 395.874,A -85,B 0,C 180,E1 -461.323,E2 -461.323} C_VEL
LIN {X 0,Y 608.542,Z 383.503,A -85,B 0,C 180,E1 -461.639,E2 -461.639} C_VEL
LIN {X 0,Y 608.575,Z 367.718,A -85,B 0,C 180,E1 -461.871,E2 -461.871} C_VEL
LIN {X 0,Y 608.547,Z 271.739,A -85,B 0,C 180,E1 -463.015,E2 -463.015} C_VEL
LIN {X 0,Y 608.459,Z 270.649,A -85,B 0,C 180,E1 -463.102,E2 -463.102} C_VEL
LIN {X 0,Y 608.495,Z 250.709,A -85,B 0,C 180,E1 -465.921,E2 -465.921} C_VEL
LIN {X 0,Y 608.518,Z 231.164,A -85,B 0,C 180,E1 -468.728,E2 -468.728} C_VEL
LIN {X 0,Y 608.55,Z 212.097,A -85,B 0,C 180,E1 -471.511,E2 -471.511} C_VEL
LIN {X 0,Y 608.478,Z 211.233,A -85,B 0,C 180,E1 -471.691,E2 -471.691} C_VEL
LIN {X 0,Y 608.445,Z 211.188,A -85,B 0,C 180,E1 -474.572,E2 -474.572} C_VEL
LIN {X 0,Y 608.487,Z 211.184,A -85,B 0,C 180,E1 -477.207,E2 -477.207} C_VEL
LIN {X 0,Y 608.469,Z 211.195,A -85,B 0,C 180,E1 -479.97,E2 -479.97} C_VEL
LIN {X 0,Y 608.451,Z 211.187,A -85,B 0,C 180,E1 -482.88,E2 -482.88} C_VEL
LIN {X 0,Y 608.436,Z 211.189,A -85,B 0,C 180,E1 -485.278,E2 -485.278} C_VEL
LIN {X 0,Y 608.469,Z 211.196,A -85,B 0,C 180,E1 -488.239,E2 -488.239} C_VEL
LIN {X 0,Y 608.435,Z 211.189,A -85,B 0,C 180,E1 -491.178,E2 -491.178} C_VEL
LIN {X 0,Y 608.469,Z 211.187,A -85,B 0,C 180,E1 -493.869,E2 -493.869} C_VEL
LIN {X 0,Y 608.465,Z 211.193,A -85,B 0,C 180,E1 -496.692,E2 -496.692} C_VEL
LIN {X 0,Y 608.441,Z 211.195,A -85,B 0,C 180,E1 -498.821,E2 -498.821} C_VEL
LIN {X 0,Y 608.461,Z 211.185,A -85,B 0,C 180,E1 -501.761,E2 -501.761} C_VEL
LIN {X 0,Y 608.452,Z 211.187,A -85,B 0,C 180,E1 -503.954,E2 -503.954} C_VEL
LIN {X 0,Y 608.453,Z 211.189,A -85,B 0,C 180,E1 -506.327,E2 -506.327} C_VEL
LIN {X 0,Y 608.452,Z 211.194,A -85,B 0,C 180,E1 -508.732,E2 -508.732} C_VEL
LIN {X 0,Y 608.454,Z 211.191,A -85,B 0,C 180,E1 -511.383,E2 -511.383} C_VEL
LIN {X 0,Y 608.429,Z 211.189,A -85,B 0,C 180,E1 -513.962,E2 -513.962} C_VEL
LIN {X 0,Y 608.454,Z 211.191,A -85,B 0,C 180,E1 -516.874,E2 -516.874} C_VEL
LIN {X 0,Y 608.442,Z 211.192,A -85,B 0,C 180,E1 -519.723,E2 -519.723} C_VEL
LIN {X 0,Y 608.428,Z 211.193,A -85,B 0,C 180,E1 -521.825,E2 -521.825} C_VEL
LIN {X 0,Y 608.461,Z 211.185,A -85,B 0,C 180,E1 -524.591,E2 -524.591} C_VEL
LIN {X 0,Y 608.476,Z 211.19,A -85,B 0,C 180,E1 -527.321,E2 -527.321} C_VEL
LIN {X 0,Y 608.435,Z 211.194,A -85,B 0,C 180,E1 -530.02,E2 -530.02} C_VEL
LIN {X 0,Y 608.429,Z 211.189,A -85,B 0,C 180,E1 -532.698,E2 -532.698} C_VEL
LIN {X 0,Y 608.46,Z 211.188,A -85,B 0,C 180,E1 -535.36,E2 -535.36} C_VEL
LIN {X 0,Y 608.462,Z 211.196,A -85,B 0,C 180,E1 -538.011,E2 -538.011} C_VEL
LIN {X 0,Y 608.447,Z 211.189,A -85,B 0,C 180,E1 -540.659,E2 -540.659} C_VEL
LIN {X 0,Y 608.457,Z 211.186,A -85,B 0,C 180,E1 -543.308,E2 -543.308} C_VEL
LIN {X 0,Y 608.487,Z 211.188,A -85,B 0,C 180,E1 -545.963,E2 -545.963} C_VEL
LIN {X 0,Y 608.438,Z 211.194,A -85,B 0,C 180,E1 -548.633,E2 -548.633} C_VEL
LIN {X 0,Y 608.436,Z 211.188,A -85,B 0,C 180,E1 -549.442,E2 -549.442} C_VEL
LIN {X 0,Y 607.778,Z 211.276,A -85,B 0,C 180,E1 -549.995,E2 -549.995} C_VEL
LIN {X 0,Y 604.936,Z 211.628,A -85,B 0,C 180,E1 -550.891,E2 -550.891} C_VEL
LIN {X 0,Y 602.527,Z 211.929,A -85,B 0,C 180,E1 -551.613,E2 -551.613} C_VEL
LIN {X 0,Y 601.488,Z 212.059,A -85,B 0,C 180,E1 -552.169,E2 -552.169} C_VEL
LIN {X 0,Y 601.401,Z 212.069,A -85,B 0,C 180,E1 -552.358,E2 -552.358} C_VEL
LIN {X 0,Y 601.415,Z 212.068,A -85,B 0,C 180,E1 -554.893,E2 -554.893} C_VEL
LIN {X 0,Y 601.417,Z 212.068,A -85,B 0,C 180,E1 -556.982,E2 -556.982} C_VEL
LIN {X 0,Y 601.385,Z 212.067,A -85,B 0,C 180,E1 -559.806,E2 -559.806} C_VEL
LIN {X 0,Y 601.445,Z 212.066,A -85,B 0,C 180,E1 -562.612,E2 -562.612} C_VEL
LIN {X 0,Y 601.388,Z 212.077,A -85,B 0,C 180,E1 -564.875,E2 -564.875} C_VEL
LIN {X 0,Y 601.401,Z 212.07,A -85,B 0,C 180,E1 -567.36,E2 -567.36} C_VEL
LIN {X 0,Y 601.392,Z 212.072,A -85,B 0,C 180,E1 -569.39,E2 -569.39} C_VEL
LIN {X 0,Y 601.386,Z 212.069,A -85,B 0,C 180,E1 -571.723,E2 -571.723} C_VEL
LIN {X 0,Y 601.406,Z 212.064,A -85,B 0,C 180,E1 -574.114,E2 -574.114} C_VEL
LIN {X 0,Y 601.388,Z 212.067,A -85,B 0,C 180,E1 -576.578,E2 -576.578} C_VEL
LIN {X 0,Y 601.42,Z 212.073,A -85,B 0,C 180,E1 -579.533,E2 -579.533} C_VEL
LIN {X 0,Y 601.398,Z 212.072,A -85,B 0,C 180,E1 -581.761,E2 -581.761} C_VEL
LIN {X 0,Y 601.39,Z 212.066,A -85,B 0,C 180,E1 -584.532,E2 -584.532} C_VEL
LIN {X 0,Y 601.423,Z 212.068,A -85,B 0,C 180,E1 -587.401,E2 -587.401} C_VEL
LIN {X 0,Y 601.404,Z 212.069,A -85,B 0,C 180,E1 -590.461,E2 -590.461} C_VEL
LIN {X 0,Y 601.462,Z 212.271,A -85,B 0,C 180,E1 -591.788,E2 -591.788} C_VEL
LIN {X 0,Y 601.508,Z 224.151,A -85,B 0,C 180,E1 -593.717,E2 -593.717} C_VEL
LIN {X 0,Y 601.478,Z 241.866,A -85,B 0,C 180,E1 -596.531,E2 -596.531} C_VEL
LIN {X 0,Y 601.429,Z 256.796,A -85,B 0,C 180,E1 -598.847,E2 -598.847} C_VEL
LIN {X 0,Y 601.639,Z 258.743,A -85,B 0,C 180,E1 -598.909,E2 -598.909} C_VEL
LIN {X 0,Y 601.609,Z 364.564,A -85,B 0,C 180,E1 -600.196,E2 -600.196} C_VEL
LIN {X 0,Y 601.574,Z 378.075,A -85,B 0,C 180,E1 -600.507,E2 -600.507} C_VEL
LIN {X 0,Y 601.555,Z 390.679,A -85,B 0,C 180,E1 -600.938,E2 -600.938} C_VEL
LIN {X 0,Y 601.539,Z 402.237,A -85,B 0,C 180,E1 -601.474,E2 -601.474} C_VEL
LIN {X 0,Y 601.464,Z 413.413,A -85,B 0,C 180,E1 -602.135,E2 -602.135} C_VEL
LIN {X 0,Y 601.469,Z 423.662,A -85,B 0,C 180,E1 -602.89,E2 -602.89} C_VEL
LIN {X 0,Y 601.419,Z 431.93,A -85,B 0,C 180,E1 -603.637,E2 -603.637} C_VEL
LIN {X 0,Y 601.417,Z 439.004,A -85,B 0,C 180,E1 -604.382,E2 -604.382} C_VEL
LIN {X 0,Y 601.401,Z 446.111,A -85,B 0,C 180,E1 -605.285,E2 -605.285} C_VEL
LIN {X 0,Y 601.36,Z 453.194,A -85,B 0,C 180,E1 -606.405,E2 -606.405} C_VEL
LIN {X 0,Y 601.349,Z 458.133,A -85,B 0,C 180,E1 -607.396,E2 -607.396} C_VEL
LIN {X 0,Y 601.34,Z 462.021,A -85,B 0,C 180,E1 -608.398,E2 -608.398} C_VEL
LIN {X 0,Y 601.343,Z 465.058,A -85,B 0,C 180,E1 -609.475,E2 -609.475} C_VEL
LIN {X 0,Y 601.327,Z 466.452,A -85,B 0,C 180,E1 -610.188,E2 -610.188} C_VEL
LIN {X 0,Y 601.339,Z 467.652,A -85,B 0,C 180,E1 -611.186,E2 -611.186} C_VEL
LIN {X 0,Y 601.323,Z 467.945,A -85,B 0,C 180,E1 -612.309,E2 -612.309} C_VEL
LIN {X 0,Y 601.327,Z 467.177,A -85,B 0,C 180,E1 -613.391,E2 -613.391} C_VEL
LIN {X 0,Y 601.321,Z 465.504,A -85,B 0,C 180,E1 -614.406,E2 -614.406} C_VEL
LIN {X 0,Y 601.348,Z 462.792,A -85,B 0,C 180,E1 -615.447,E2 -615.447} C_VEL
LIN {X 0,Y 601.339,Z 459.031,A -85,B 0,C 180,E1 -616.482,E2 -616.482} C_VEL
LIN {X 0,Y 601.37,Z 454.119,A -85,B 0,C 180,E1 -617.514,E2 -617.514} C_VEL
LIN {X 0,Y 601.38,Z 447.931,A -85,B 0,C 180,E1 -618.541,E2 -618.541} C_VEL
LIN {X 0,Y 601.395,Z 440.258,A -85,B 0,C 180,E1 -619.564,E2 -619.564} C_VEL
LIN {X 0,Y 601.424,Z 432.318,A -85,B 0,C 180,E1 -620.414,E2 -620.414} C_VEL
LIN {X 0,Y 601.444,Z 423.951,A -85,B 0,C 180,E1 -621.178,E2 -621.178} C_VEL
LIN {X 0,Y 601.438,Z 413.664,A -85,B 0,C 180,E1 -621.939,E2 -621.939} C_VEL
LIN {X 0,Y 601.493,Z 402.266,A -85,B 0,C 180,E1 -622.615,E2 -622.615} C_VEL
LIN {X 0,Y 601.549,Z 390.999,A -85,B 0,C 180,E1 -623.139,E2 -623.139} C_VEL
LIN {X 0,Y 601.6,Z 378.07,A -85,B 0,C 180,E1 -623.583,E2 -623.583} C_VEL
LIN {X 0,Y 601.623,Z 364.637,A -85,B 0,C 180,E1 -623.892,E2 -623.892} C_VEL
LIN {X 0,Y 601.502,Z 257.531,A -85,B 0,C 180,E1 -625.203,E2 -625.203} C_VEL
LIN {X 0,Y 601.423,Z 256.253,A -85,B 0,C 180,E1 -625.308,E2 -625.308} C_VEL
LIN {X 0,Y 601.446,Z 239.139,A -85,B 0,C 180,E1 -627.991,E2 -627.991} C_VEL
LIN {X 0,Y 601.468,Z 223.355,A -85,B 0,C 180,E1 -630.502,E2 -630.502} C_VEL
LIN {X 0,Y 601.481,Z 212.266,A -85,B 0,C 180,E1 -632.302,E2 -632.302} C_VEL
LIN {X 0,Y 601.443,Z 212.06,A -85,B 0,C 180,E1 -635.364,E2 -635.364} C_VEL
LIN {X 0,Y 601.419,Z 212.067,A -85,B 0,C 180,E1 -638.061,E2 -638.061} C_VEL
LIN {X 0,Y 601.447,Z 212.062,A -85,B 0,C 180,E1 -641.052,E2 -641.052} C_VEL
LIN {X 0,Y 601.405,Z 212.064,A -85,B 0,C 180,E1 -643.516,E2 -643.516} C_VEL
LIN {X 0,Y 601.44,Z 212.063,A -85,B 0,C 180,E1 -646.287,E2 -646.287} C_VEL
LIN {X 0,Y 601.401,Z 212.071,A -85,B 0,C 180,E1 -649.099,E2 -649.099} C_VEL
LIN {X 0,Y 601.404,Z 212.064,A -85,B 0,C 180,E1 -651.959,E2 -651.959} C_VEL
LIN {X 0,Y 601.42,Z 212.063,A -85,B 0,C 180,E1 -654.302,E2 -654.302} C_VEL
LIN {X 0,Y 601.439,Z 212.069,A -85,B 0,C 180,E1 -657.111,E2 -657.111} C_VEL
LIN {X 0,Y 601.449,Z 212.059,A -85,B 0,C 180,E1 -660.162,E2 -660.162} C_VEL
LIN {X 0,Y 601.429,Z 212.071,A -85,B 0,C 180,E1 -663.313,E2 -663.313} C_VEL
LIN {X 0,Y 601.414,Z 212.064,A -85,B 0,C 180,E1 -666.271,E2 -666.271} C_VEL
LIN {X 0,Y 601.413,Z 212.066,A -85,B 0,C 180,E1 -669.126,E2 -669.126} C_VEL
LIN {X 0,Y 601.408,Z 212.075,A -85,B 0,C 180,E1 -671.766,E2 -671.766} C_VEL
LIN {X 0,Y 601.42,Z 212.063,A -85,B 0,C 180,E1 -674.542,E2 -674.542} C_VEL
LIN {X 0,Y 601.413,Z 212.065,A -85,B 0,C 180,E1 -677.409,E2 -677.409} C_VEL
LIN {X 0,Y 601.428,Z 212.065,A -85,B 0,C 180,E1 -680.465,E2 -680.465} C_VEL
LIN {X 0,Y 601.401,Z 212.064,A -85,B 0,C 180,E1 -683.423,E2 -683.423} C_VEL
LIN {X 0,Y 601.422,Z 212.068,A -85,B 0,C 180,E1 -686.065,E2 -686.065} C_VEL
LIN {X 0,Y 601.423,Z 212.071,A -85,B 0,C 180,E1 -688.544,E2 -688.544} C_VEL
LIN {X 0,Y 601.427,Z 212.061,A -85,B 0,C 180,E1 -691.378,E2 -691.378} C_VEL
LIN {X 0,Y 601.395,Z 212.064,A -85,B 0,C 180,E1 -693.641,E2 -693.641} C_VEL
LIN {X 0,Y 601.408,Z 212.072,A -85,B 0,C 180,E1 -696.594,E2 -696.594} C_VEL
LIN {X 0,Y 601.425,Z 212.063,A -85,B 0,C 180,E1 -699.482,E2 -699.482} C_VEL
LIN {X 0,Y 601.387,Z 212.067,A -85,B 0,C 180,E1 -702.315,E2 -702.315} C_VEL
LIN {X 0,Y 601.405,Z 212.064,A -85,B 0,C 180,E1 -704.412,E2 -704.412} C_VEL
LIN {X 0,Y 601.414,Z 212.074,A -85,B 0,C 180,E1 -707.175,E2 -707.175} C_VEL
LIN {X 0,Y 601.437,Z 212.062,A -85,B 0,C 180,E1 -709.909,E2 -709.909} C_VEL
LIN {X 0,Y 601.43,Z 212.062,A -85,B 0,C 180,E1 -712.618,E2 -712.618} C_VEL
LIN {X 0,Y 601.424,Z 212.07,A -85,B 0,C 180,E1 -715.311,E2 -715.311} C_VEL
LIN {X 0,Y 601.423,Z 212.065,A -85,B 0,C 180,E1 -717.994,E2 -717.994} C_VEL
LIN {X 0,Y 601.447,Z 212.058,A -85,B 0,C 180,E1 -720.673,E2 -720.673} C_VEL
LIN {X 0,Y 601.414,Z 212.066,A -85,B 0,C 180,E1 -723.352,E2 -723.352} C_VEL
LIN {X 0,Y 601.421,Z 212.071,A -85,B 0,C 180,E1 -726.04,E2 -726.04} C_VEL
LIN {X 0,Y 601.412,Z 212.063,A -85,B 0,C 180,E1 -728.741,E2 -728.741} C_VEL
LIN {X 0,Y 601.413,Z 212.063,A -85,B 0,C 180,E1 -731.461,E2 -731.461} C_VEL
LIN {X 0,Y 601.421,Z 212.073,A -85,B 0,C 180,E1 -734.208,E2 -734.208} C_VEL
LIN {X 0,Y 601.433,Z 212.062,A -85,B 0,C 180,E1 -736.988,E2 -736.988} C_VEL
LIN {X 0,Y 601.401,Z 212.065,A -85,B 0,C 180,E1 -739.812,E2 -739.812} C_VEL
LIN {X 0,Y 601.42,Z 212.073,A -85,B 0,C 180,E1 -742.608,E2 -742.608} C_VEL
LIN {X 0,Y 601.4,Z 212.072,A -85,B 0,C 180,E1 -744.881,E2 -744.881} C_VEL
LIN {X 0,Y 601.414,Z 212.065,A -85,B 0,C 180,E1 -747.363,E2 -747.363} C_VEL
LIN {X 0,Y 601.42,Z 212.064,A -85,B 0,C 180,E1 -749.395,E2 -749.395} C_VEL
LIN {X 0,Y 601.399,Z 212.065,A -85,B 0,C 180,E1 -751.729,E2 -751.729} C_VEL
LIN {X 0,Y 601.418,Z 212.063,A -85,B 0,C 180,E1 -754.121,E2 -754.121} C_VEL
LIN {X 0,Y 601.4,Z 212.067,A -85,B 0,C 180,E1 -756.585,E2 -756.585} C_VEL
LIN {X 0,Y 601.408,Z 212.073,A -85,B 0,C 180,E1 -759.129,E2 -759.129} C_VEL
LIN {X 0,Y 601.431,Z 212.064,A -85,B 0,C 180,E1 -761.766,E2 -761.766} C_VEL
LIN {X 0,Y 601.403,Z 212.063,A -85,B 0,C 180,E1 -764.534,E2 -764.534} C_VEL
LIN {X 0,Y 601.414,Z 212.071,A -85,B 0,C 180,E1 -767.411,E2 -767.411} C_VEL
LIN {X 0,Y 601.404,Z 212.069,A -85,B 0,C 180,E1 -770.005,E2 -770.005} C_VEL
LIN {X 0,Y 601.437,Z 212.06,A -85,B 0,C 180,E1 -772.619,E2 -772.619} C_VEL
LIN {X 0,Y 601.396,Z 212.066,A -85,B 0,C 180,E1 -775.067,E2 -775.067} C_VEL
LIN {X 0,Y 601.417,Z 212.066,A -85,B 0,C 180,E1 -777.484,E2 -777.484} C_VEL
LIN {X 0,Y 601.411,Z 212.071,A -85,B 0,C 180,E1 -779.856,E2 -779.856} C_VEL
LIN {X 0,Y 601.456,Z 212.059,A -85,B 0,C 180,E1 -782.89,E2 -782.89} C_VEL
LIN {X 0,Y 601.408,Z 212.067,A -85,B 0,C 180,E1 -785.715,E2 -785.715} C_VEL
LIN {X 0,Y 601.451,Z 212.243,A -85,B 0,C 180,E1 -788.223,E2 -788.223} C_VEL
LIN {X 0,Y 601.606,Z 219.103,A -85,B 0,C 180,E1 -789.271,E2 -789.271} C_VEL
LIN {X 0,Y 601.529,Z 237.439,A -85,B 0,C 180,E1 -791.964,E2 -791.964} C_VEL
LIN {X 0,Y 601.45,Z 255.539,A -85,B 0,C 180,E1 -794.584,E2 -794.584} C_VEL
LIN {X 0,Y 601.461,Z 271.287,A -85,B 0,C 180,E1 -796.808,E2 -796.808} C_VEL
LIN {X 0,Y 601.67,Z 274.744,A -85,B 0,C 180,E1 -796.877,E2 -796.877} C_VEL
LIN {X 0,Y 601.62,Z 378.962,A -85,B 0,C 180,E1 -798.14,E2 -798.14} C_VEL
LIN {X 0,Y 601.591,Z 392.227,A -85,B 0,C 180,E1 -798.438,E2 -798.438} C_VEL
LIN {X 0,Y 601.55,Z 403.937,A -85,B 0,C 180,E1 -798.827,E2 -798.827} C_VEL
LIN {X 0,Y 601.531,Z 414.93,A -85,B 0,C 180,E1 -799.311,E2 -799.311} C_VEL
LIN {X 0,Y 601.462,Z 425.585,A -85,B 0,C 180,E1 -799.906,E2 -799.906} C_VEL
LIN {X 0,Y 601.447,Z 436.479,A -85,B 0,C 180,E1 -800.67,E2 -800.67} C_VEL
LIN {X 0,Y 601.423,Z 445.321,A -85,B 0,C 180,E1 -801.432,E2 -801.432} C_VEL
LIN {X 0,Y 601.396,Z 453.48,A -85,B 0,C 180,E1 -802.277,E2 -802.277} C_VEL
LIN {X 0,Y 601.382,Z 461.472,A -85,B 0,C 180,E1 -803.289,E2 -803.289} C_VEL
LIN {X 0,Y 601.372,Z 467.867,A -85,B 0,C 180,E1 -804.299,E2 -804.299} C_VEL
LIN {X 0,Y 601.336,Z 472.951,A -85,B 0,C 180,E1 -805.308,E2 -805.308} C_VEL
LIN {X 0,Y 601.367,Z 476.897,A -85,B 0,C 180,E1 -806.315,E2 -806.315} C_VEL
LIN {X 0,Y 601.325,Z 479.81,A -85,B 0,C 180,E1 -807.321,E2 -807.321} C_VEL
LIN {X 0,Y 601.341,Z 481.202,A -85,B 0,C 180,E1 -807.991,E2 -807.991} C_VEL
LIN {X 0,Y 601.339,Z 482.784,A -85,B 0,C 180,E1 -809.331,E2 -809.331} C_VEL
LIN {X 0,Y 601.335,Z 483,A -85,B 0,C 180,E1 -810,E2 -810} C_VEL
LIN {X 0,Y 601.347,Z 482.184,A -85,B 0,C 180,E1 -811.34,E2 -811.34} C_VEL
LIN {X 0,Y 601.341,Z 481.202,A -85,B 0,C 180,E1 -812.01,E2 -812.01} C_VEL
LIN {X 0,Y 601.325,Z 479.809,A -85,B 0,C 180,E1 -812.68,E2 -812.68} C_VEL
LIN {X 0,Y 601.367,Z 476.895,A -85,B 0,C 180,E1 -813.686,E2 -813.686} C_VEL
LIN {X 0,Y 601.336,Z 472.949,A -85,B 0,C 180,E1 -814.693,E2 -814.693} C_VEL
LIN {X 0,Y 601.372,Z 466.876,A -85,B 0,C 180,E1 -815.869,E2 -815.869} C_VEL
LIN {X 0,Y 601.382,Z 460.234,A -85,B 0,C 180,E1 -816.88,E2 -816.88} C_VEL
LIN {X 0,Y 601.401,Z 451.988,A -85,B 0,C 180,E1 -817.892,E2 -817.892} C_VEL
LIN {X 0,Y 601.435,Z 441.597,A -85,B 0,C 180,E1 -818.907,E2 -818.907} C_VEL
LIN {X 0,Y 601.472,Z 430.745,A -85,B 0,C 180,E1 -819.755,E2 -819.755} C_VEL
LIN {X 0,Y 601.495,Z 419.772,A -85,B 0,C 180,E1 -820.434,E2 -820.434} C_VEL
LIN {X 0,Y 601.552,Z 407.656,A -85,B 0,C 180,E1 -821.023,E2 -821.023} C_VEL
LIN {X 0,Y 601.579,Z 395.871,A -85,B 0,C 180,E1 -821.455,E2 -821.455} C_VEL
LIN {X 0,Y 601.609,Z 383.501,A -85,B 0,C 180,E1 -821.775,E2 -821.775} C_VEL
LIN {X 0,Y 601.643,Z 367.718,A -85,B 0,C 180,E1 -822.01,E2 -822.01} C_VEL
LIN {X 0,Y 601.574,Z 272.205,A -85,B 0,C 180,E1 -823.158,E2 -823.158} C_VEL
LIN {X 0,Y 601.453,Z 271.005,A -85,B 0,C 180,E1 -823.214,E2 -823.214} C_VEL
LIN {X 0,Y 601.485,Z 251.915,A -85,B 0,C 180,E1 -825.937,E2 -825.937} C_VEL
LIN {X 0,Y 601.532,Z 233.419,A -85,B 0,C 180,E1 -828.623,E2 -828.623} C_VEL
LIN {X 0,Y 601.647,Z 214.51,A -85,B 0,C 180,E1 -831.41,E2 -831.41} C_VEL
LIN {X 0,Y 601.437,Z 212.107,A -85,B 0,C 180,E1 -831.823,E2 -831.823} C_VEL
LIN {X 0,Y 601.408,Z 212.067,A -85,B 0,C 180,E1 -834.285,E2 -834.285} C_VEL
LIN {X 0,Y 601.457,Z 212.059,A -85,B 0,C 180,E1 -837.111,E2 -837.111} C_VEL
LIN {X 0,Y 601.411,Z 212.07,A -85,B 0,C 180,E1 -840.165,E2 -840.165} C_VEL
LIN {X 0,Y 601.411,Z 212.064,A -85,B 0,C 180,E1 -842.712,E2 -842.712} C_VEL
LIN {X 0,Y 601.385,Z 212.067,A -85,B 0,C 180,E1 -845.109,E2 -845.109} C_VEL
LIN {X 0,Y 601.438,Z 212.061,A -85,B 0,C 180,E1 -847.419,E2 -847.419} C_VEL
LIN {X 0,Y 601.406,Z 212.07,A -85,B 0,C 180,E1 -849.995,E2 -849.995} C_VEL
LIN {X 0,Y 601.411,Z 212.069,A -85,B 0,C 180,E1 -852.67,E2 -852.67} C_VEL
LIN {X 0,Y 601.407,Z 212.064,A -85,B 0,C 180,E1 -855.479,E2 -855.479} C_VEL
LIN {X 0,Y 601.428,Z 212.069,A -85,B 0,C 180,E1 -858.406,E2 -858.406} C_VEL
LIN {X 0,Y 601.401,Z 212.072,A -85,B 0,C 180,E1 -860.871,E2 -860.871} C_VEL
LIN {X 0,Y 601.395,Z 212.067,A -85,B 0,C 180,E1 -863.415,E2 -863.415} C_VEL
LIN {X 0,Y 601.421,Z 212.063,A -85,B 0,C 180,E1 -866.066,E2 -866.066} C_VEL
LIN {X 0,Y 601.405,Z 212.074,A -85,B 0,C 180,E1 -869.055,E2 -869.055} C_VEL
LIN {X 0,Y 601.414,Z 212.068,A -85,B 0,C 180,E1 -871.37,E2 -871.37} C_VEL
LIN {X 0,Y 601.393,Z 212.068,A -85,B 0,C 180,E1 -873.634,E2 -873.634} C_VEL
LIN {X 0,Y 601.408,Z 212.065,A -85,B 0,C 180,E1 -875.855,E2 -875.855} C_VEL
LIN {X 0,Y 601.407,Z 212.067,A -85,B 0,C 180,E1 -878.759,E2 -878.759} C_VEL
LIN {X 0,Y 601.396,Z 212.073,A -85,B 0,C 180,E1 -881.605,E2 -881.605} C_VEL
LIN {X 0,Y 601.428,Z 212.068,A -85,B 0,C 180,E1 -883.71,E2 -883.71} C_VEL
LIN {X 0,Y 601.399,Z 212.065,A -85,B 0,C 180,E1 -886.481,E2 -886.481} C_VEL
LIN {X 0,Y 601.423,Z 212.065,A -85,B 0,C 180,E1 -889.221,E2 -889.221} C_VEL
LIN {X 0,Y 601.409,Z 212.072,A -85,B 0,C 180,E1 -891.936,E2 -891.936} C_VEL
LIN {X 0,Y 601.399,Z 212.065,A -85,B 0,C 180,E1 -894.633,E2 -894.633} C_VEL
LIN {X 0,Y 601.442,Z 212.061,A -85,B 0,C 180,E1 -897.318,E2 -897.318} C_VEL
LIN {X 0,Y 601.447,Z 212.07,A -85,B 0,C 180,E1 -899.997,E2 -899.997} C_VEL
LIN {X 0,Y 601.415,Z 212.065,A -85,B 0,C 180,E1 -902.676,E2 -902.676} C_VEL
LIN {X 0,Y 601.408,Z 212.064,A -85,B 0,C 180,E1 -905.361,E2 -905.361} C_VEL
LIN {X 0,Y 601.437,Z 212.066,A -85,B 0,C 180,E1 -908.057,E2 -908.057} C_VEL
LIN {X 0,Y 601.396,Z 212.067,A -85,B 0,C 180,E1 -910.998,E2 -910.998} C_VEL
LIN {X 0,Y 601.401,Z 212.069,A -85,B 0,C 180,E1 -912.358,E2 -912.358} C_VEL
LIN {X 0,Y 600.73,Z 212.154,A -85,B 0,C 180,E1 -912.917,E2 -912.917} C_VEL
LIN {X 0,Y 597.878,Z 212.508,A -85,B 0,C 180,E1 -913.825,E2 -913.825} C_VEL
LIN {X 0,Y 595.469,Z 212.815,A -85,B 0,C 180,E1 -914.555,E2 -914.555} C_VEL
LIN {X 0,Y 594.431,Z 212.936,A -85,B 0,C 180,E1 -915.119,E2 -915.119} C_VEL
LIN {X 0,Y 594.345,Z 212.944,A -85,B 0,C 180,E1 -915.31,E2 -915.31} C_VEL
LIN {X 0,Y 594.373,Z 212.943,A -85,B 0,C 180,E1 -917.19,E2 -917.19} C_VEL
LIN {X 0,Y 594.362,Z 212.943,A -85,B 0,C 180,E1 -920.05,E2 -920.05} C_VEL
LIN {X 0,Y 594.36,Z 212.952,A -85,B 0,C 180,E1 -922.963,E2 -922.963} C_VEL
LIN {X 0,Y 594.353,Z 212.948,A -85,B 0,C 180,E1 -925.189,E2 -925.189} C_VEL
LIN {X 0,Y 594.366,Z 212.944,A -85,B 0,C 180,E1 -927.523,E2 -927.523} C_VEL
LIN {X 0,Y 594.351,Z 212.943,A -85,B 0,C 180,E1 -930.322,E2 -930.322} C_VEL
LIN {X 0,Y 594.355,Z 212.949,A -85,B 0,C 180,E1 -932.946,E2 -932.946} C_VEL
LIN {X 0,Y 594.356,Z 212.952,A -85,B 0,C 180,E1 -935.403,E2 -935.403} C_VEL
LIN {X 0,Y 594.356,Z 212.945,A -85,B 0,C 180,E1 -937.937,E2 -937.937} C_VEL
LIN {X 0,Y 594.358,Z 212.943,A -85,B 0,C 180,E1 -940.82,E2 -940.82} C_VEL
LIN {X 0,Y 594.35,Z 212.95,A -85,B 0,C 180,E1 -943.838,E2 -943.838} C_VEL
LIN {X 0,Y 594.34,Z 212.945,A -85,B 0,C 180,E1 -946.698,E2 -946.698} C_VEL
LIN {X 0,Y 594.37,Z 212.946,A -85,B 0,C 180,E1 -949.433,E2 -949.433} C_VEL
LIN {X 0,Y 594.423,Z 213.165,A -85,B 0,C 180,E1 -951.685,E2 -951.685} C_VEL
LIN {X 0,Y 594.542,Z 222.6,A -85,B 0,C 180,E1 -953.243,E2 -953.243} C_VEL
LIN {X 0,Y 594.459,Z 239.999,A -85,B 0,C 180,E1 -956.044,E2 -956.044} C_VEL
LIN {X 0,Y 594.399,Z 256.662,A -85,B 0,C 180,E1 -958.676,E2 -958.676} C_VEL
LIN {X 0,Y 594.575,Z 258.382,A -85,B 0,C 180,E1 -958.745,E2 -958.745} C_VEL
LIN {X 0,Y 594.682,Z 364.61,A -85,B 0,C 180,E1 -960.057,E2 -960.057} C_VEL
LIN {X 0,Y 594.626,Z 377.689,A -85,B 0,C 180,E1 -960.359,E2 -960.359} C_VEL
LIN {X 0,Y 594.595,Z 390.136,A -85,B 0,C 180,E1 -960.785,E2 -960.785} C_VEL
LIN {X 0,Y 594.523,Z 401.336,A -85,B 0,C 180,E1 -961.299,E2 -961.299} C_VEL
LIN {X 0,Y 594.463,Z 412.647,A -85,B 0,C 180,E1 -961.965,E2 -961.965} C_VEL
LIN {X 0,Y 594.435,Z 423.075,A -85,B 0,C 180,E1 -962.733,E2 -962.733} C_VEL
LIN {X 0,Y 594.374,Z 431.429,A -85,B 0,C 180,E1 -963.485,E2 -963.485} C_VEL
LIN {X 0,Y 594.347,Z 440.211,A -85,B 0,C 180,E1 -964.431,E2 -964.431} C_VEL
LIN {X 0,Y 594.301,Z 448.447,A -85,B 0,C 180,E1 -965.55,E2 -965.55} C_VEL
LIN {X 0,Y 594.266,Z 454.914,A -85,B 0,C 180,E1 -966.66,E2 -966.66} C_VEL
LIN {X 0,Y 594.265,Z 459.892,A -85,B 0,C 180,E1 -967.763,E2 -967.763} C_VEL
LIN {X 0,Y 594.256,Z 464.201,A -85,B 0,C 180,E1 -969.099,E2 -969.099} C_VEL
LIN {X 0,Y 594.224,Z 466.084,A -85,B 0,C 180,E1 -969.941,E2 -969.941} C_VEL
LIN {X 0,Y 594.251,Z 467.594,A -85,B 0,C 180,E1 -971.091,E2 -971.091} C_VEL
LIN {X 0,Y 594.214,Z 467.996,A -85,B 0,C 180,E1 -972.091,E2 -972.091} C_VEL
LIN {X 0,Y 594.234,Z 467.285,A -85,B 0,C 180,E1 -973.313,E2 -973.313} C_VEL
LIN {X 0,Y 594.245,Z 465.963,A -85,B 0,C 180,E1 -974.216,E2 -974.216} C_VEL
LIN {X 0,Y 594.253,Z 463.465,A -85,B 0,C 180,E1 -975.269,E2 -975.269} C_VEL
LIN {X 0,Y 594.254,Z 459.93,A -85,B 0,C 180,E1 -976.318,E2 -976.318} C_VEL
LIN {X 0,Y 594.27,Z 455.271,A -85,B 0,C 180,E1 -977.362,E2 -977.362} C_VEL
LIN {X 0,Y 594.319,Z 448.148,A -85,B 0,C 180,E1 -978.585,E2 -978.585} C_VEL
LIN {X 0,Y 594.319,Z 440.605,A -85,B 0,C 180,E1 -979.611,E2 -979.611} C_VEL
LIN {X 0,Y 594.362,Z 432.763,A -85,B 0,C 180,E1 -980.471,E2 -980.471} C_VEL
LIN {X 0,Y 594.411,Z 423.424,A -85,B 0,C 180,E1 -981.329,E2 -981.329} C_VEL
LIN {X 0,Y 594.453,Z 413.017,A -85,B 0,C 180,E1 -982.1,E2 -982.1} C_VEL
LIN {X 0,Y 594.498,Z 402.73,A -85,B 0,C 180,E1 -982.716,E2 -982.716} C_VEL
LIN {X 0,Y 594.577,Z 391.262,A -85,B 0,C 180,E1 -983.26,E2 -983.26} C_VEL
LIN {X 0,Y 594.605,Z 377.896,A -85,B 0,C 180,E1 -983.725,E2 -983.725} C_VEL
LIN {X 0,Y 594.672,Z 365.225,A -85,B 0,C 180,E1 -984.022,E2 -984.022} C_VEL
LIN {X 0,Y 594.668,Z 328.612,A -85,B 0,C 180,E1 -984.49,E2 -984.49} C_VEL
LIN {X 0,Y 594.642,Z 258.651,A -85,B 0,C 180,E1 -985.339,E2 -985.339} C_VEL
LIN {X 0,Y 594.412,Z 256.79,A -85,B 0,C 180,E1 -985.401,E2 -985.401} C_VEL
LIN {X 0,Y 594.445,Z 240.493,A -85,B 0,C 180,E1 -987.967,E2 -987.967} C_VEL
LIN {X 0,Y 594.51,Z 223.655,A -85,B 0,C 180,E1 -990.677,E2 -990.677} C_VEL
LIN {X 0,Y 594.452,Z 213.332,A -85,B 0,C 180,E1 -992.371,E2 -992.371} C_VEL
LIN {X 0,Y 594.395,Z 212.96,A -85,B 0,C 180,E1 -992.541,E2 -992.541} C_VEL
LIN {X 0,Y 594.402,Z 212.937,A -85,B 0,C 180,E1 -995.427,E2 -995.427} C_VEL
LIN {X 0,Y 594.394,Z 212.944,A -85,B 0,C 180,E1 -998.157,E2 -998.157} C_VEL
LIN {X 0,Y 594.419,Z 212.937,A -85,B 0,C 180,E1 -1001.117,E2 -1001.117} C_VEL
LIN {X 0,Y 594.384,Z 212.942,A -85,B 0,C 180,E1 -1004.194,E2 -1004.194} C_VEL
LIN {X 0,Y 594.363,Z 212.945,A -85,B 0,C 180,E1 -1007.194,E2 -1007.194} C_VEL
LIN {X 0,Y 594.357,Z 212.941,A -85,B 0,C 180,E1 -1010.054,E2 -1010.054} C_VEL
LIN {X 0,Y 594.378,Z 212.95,A -85,B 0,C 180,E1 -1012.966,E2 -1012.966} C_VEL
LIN {X 0,Y 594.359,Z 212.95,A -85,B 0,C 180,E1 -1015.193,E2 -1015.193} C_VEL
LIN {X 0,Y 594.36,Z 212.946,A -85,B 0,C 180,E1 -1017.533,E2 -1017.533} C_VEL
LIN {X 0,Y 594.387,Z 212.938,A -85,B 0,C 180,E1 -1020.339,E2 -1020.339} C_VEL
LIN {X 0,Y 594.384,Z 212.942,A -85,B 0,C 180,E1 -1022.949,E2 -1022.949} C_VEL
LIN {X 0,Y 594.361,Z 212.951,A -85,B 0,C 180,E1 -1025.408,E2 -1025.408} C_VEL
LIN {X 0,Y 594.365,Z 212.947,A -85,B 0,C 180,E1 -1027.942,E2 -1027.942} C_VEL
LIN {X 0,Y 594.37,Z 212.94,A -85,B 0,C 180,E1 -1030.829,E2 -1030.829} C_VEL
LIN {X 0,Y 594.352,Z 212.944,A -85,B 0,C 180,E1 -1033.3,E2 -1033.3} C_VEL
LIN {X 0,Y 594.362,Z 212.949,A -85,B 0,C 180,E1 -1036.16,E2 -1036.16} C_VEL
LIN {X 0,Y 594.369,Z 212.943,A -85,B 0,C 180,E1 -1038.542,E2 -1038.542} C_VEL
LIN {X 0,Y 594.37,Z 212.939,A -85,B 0,C 180,E1 -1041.297,E2 -1041.297} C_VEL
LIN {X 0,Y 594.376,Z 212.942,A -85,B 0,C 180,E1 -1043.763,E2 -1043.763} C_VEL
LIN {X 0,Y 594.369,Z 212.95,A -85,B 0,C 180,E1 -1046.244,E2 -1046.244} C_VEL
LIN {X 0,Y 594.372,Z 212.947,A -85,B 0,C 180,E1 -1048.655,E2 -1048.655} C_VEL
LIN {X 0,Y 594.375,Z 212.941,A -85,B 0,C 180,E1 -1051.043,E2 -1051.043} C_VEL
LIN {X 0,Y 594.377,Z 212.939,A -85,B 0,C 180,E1 -1053.305,E2 -1053.305} C_VEL
LIN {X 0,Y 594.377,Z 212.943,A -85,B 0,C 180,E1 -1056.3,E2 -1056.3} C_VEL
LIN {X 0,Y 594.396,Z 212.942,A -85,B 0,C 180,E1 -1059.228,E2 -1059.228} C_VEL
LIN {X 0,Y 594.368,Z 212.94,A -85,B 0,C 180,E1 -1062.1,E2 -1062.1} C_VEL
LIN {X 0,Y 594.36,Z 212.94,A -85,B 0,C 180,E1 -1064.223,E2 -1064.223} C_VEL
LIN {X 0,Y 594.36,Z 212.949,A -85,B 0,C 180,E1 -1067.021,E2 -1067.021} C_VEL
LIN {X 0,Y 594.396,Z 212.94,A -85,B 0,C 180,E1 -1069.788,E2 -1069.788} C_VEL
LIN {X 0,Y 594.385,Z 212.939,A -85,B 0,C 180,E1 -1072.53,E2 -1072.53} C_VEL
LIN {X 0,Y 594.392,Z 212.944,A -85,B 0,C 180,E1 -1075.256,E2 -1075.256} C_VEL
LIN {X 0,Y 594.393,Z 212.94,A -85,B 0,C 180,E1 -1077.97,E2 -1077.97} C_VEL
LIN {X 0,Y 594.418,Z 212.934,A -85,B 0,C 180,E1 -1080.68,E2 -1080.68} C_VEL
LIN {X 0,Y 594.367,Z 212.945,A -85,B 0,C 180,E1 -1083.392,E2 -1083.392} C_VEL
LIN {X 0,Y 594.374,Z 212.947,A -85,B 0,C 180,E1 -1086.112,E2 -1086.112} C_VEL
LIN {X 0,Y 594.378,Z 212.938,A -85,B 0,C 180,E1 -1088.845,E2 -1088.845} C_VEL
LIN {X 0,Y 594.38,Z 212.94,A -85,B 0,C 180,E1 -1091.599,E2 -1091.599} C_VEL
LIN {X 0,Y 594.391,Z 212.947,A -85,B 0,C 180,E1 -1094.379,E2 -1094.379} C_VEL
LIN {X 0,Y 594.389,Z 212.938,A -85,B 0,C 180,E1 -1097.196,E2 -1097.196} C_VEL
LIN {X 0,Y 594.373,Z 212.943,A -85,B 0,C 180,E1 -1100.056,E2 -1100.056} C_VEL
LIN {X 0,Y 594.359,Z 212.946,A -85,B 0,C 180,E1 -1102.97,E2 -1102.97} C_VEL
LIN {X 0,Y 594.375,Z 212.943,A -85,B 0,C 180,E1 -1105.195,E2 -1105.195} C_VEL
LIN {X 0,Y 594.373,Z 212.941,A -85,B 0,C 180,E1 -1107.525,E2 -1107.525} C_VEL
LIN {X 0,Y 594.372,Z 212.941,A -85,B 0,C 180,E1 -1110.327,E2 -1110.327} C_VEL
LIN {X 0,Y 594.379,Z 212.951,A -85,B 0,C 180,E1 -1112.952,E2 -1112.952} C_VEL
LIN {X 0,Y 594.352,Z 212.948,A -85,B 0,C 180,E1 -1115.411,E2 -1115.411} C_VEL
LIN {X 0,Y 594.386,Z 212.939,A -85,B 0,C 180,E1 -1117.943,E2 -1117.943} C_VEL
LIN {X 0,Y 594.377,Z 212.943,A -85,B 0,C 180,E1 -1120.823,E2 -1120.823} C_VEL
LIN {X 0,Y 594.365,Z 212.943,A -85,B 0,C 180,E1 -1123.84,E2 -1123.84} C_VEL
LIN {X 0,Y 594.355,Z 212.941,A -85,B 0,C 180,E1 -1126.7,E2 -1126.7} C_VEL
LIN {X 0,Y 594.366,Z 212.949,A -85,B 0,C 180,E1 -1129.433,E2 -1129.433} C_VEL
LIN {X 0,Y 594.392,Z 212.939,A -85,B 0,C 180,E1 -1132.393,E2 -1132.393} C_VEL
LIN {X 0,Y 594.374,Z 212.944,A -85,B 0,C 180,E1 -1135.42,E2 -1135.42} C_VEL
LIN {X 0,Y 594.38,Z 212.944,A -85,B 0,C 180,E1 -1138.359,E2 -1138.359} C_VEL
LIN {X 0,Y 594.38,Z 212.94,A -85,B 0,C 180,E1 -1141.044,E2 -1141.044} C_VEL
LIN {X 0,Y 594.386,Z 212.939,A -85,B 0,C 180,E1 -1143.301,E2 -1143.301} C_VEL
LIN {X 0,Y 594.376,Z 212.952,A -85,B 0,C 180,E1 -1146.296,E2 -1146.296} C_VEL
LIN {X 0,Y 594.394,Z 213.137,A -85,B 0,C 180,E1 -1148.088,E2 -1148.088} C_VEL
LIN {X 0,Y 594.693,Z 216.845,A -85,B 0,C 180,E1 -1148.679,E2 -1148.679} C_VEL
LIN {X 0,Y 594.574,Z 236.233,A -85,B 0,C 180,E1 -1151.568,E2 -1151.568} C_VEL
LIN {X 0,Y 594.486,Z 254.332,A -85,B 0,C 180,E1 -1154.223,E2 -1154.223} C_VEL
LIN {X 0,Y 594.43,Z 271.279,A -85,B 0,C 180,E1 -1156.649,E2 -1156.649} C_VEL
LIN {X 0,Y 594.768,Z 274.744,A -85,B 0,C 180,E1 -1156.722,E2 -1156.722} C_VEL
LIN {X 0,Y 594.673,Z 378.962,A -85,B 0,C 180,E1 -1157.999,E2 -1157.999} C_VEL
LIN {X 0,Y 594.64,Z 392.228,A -85,B 0,C 180,E1 -1158.301,E2 -1158.301} C_VEL
LIN {X 0,Y 594.588,Z 405.382,A -85,B 0,C 180,E1 -1158.75,E2 -1158.75} C_VEL
LIN {X 0,Y 594.537,Z 416.637,A -85,B 0,C 180,E1 -1159.27,E2 -1159.27} C_VEL
LIN {X 0,Y 594.455,Z 428.205,A -85,B 0,C 180,E1 -1159.958,E2 -1159.958} C_VEL
LIN {X 0,Y 594.413,Z 438.6,A -85,B 0,C 180,E1 -1160.73,E2 -1160.73} C_VEL
LIN {X 0,Y 594.349,Z 447.035,A -85,B 0,C 180,E1 -1161.5,E2 -1161.5} C_VEL
LIN {X 0,Y 594.347,Z 454.963,A -85,B 0,C 180,E1 -1162.356,E2 -1162.356} C_VEL
LIN {X 0,Y 594.281,Z 462.831,A -85,B 0,C 180,E1 -1163.411,E2 -1163.411} C_VEL
LIN {X 0,Y 594.289,Z 469.682,A -85,B 0,C 180,E1 -1164.572,E2 -1164.572} C_VEL
LIN {X 0,Y 594.27,Z 474.372,A -85,B 0,C 180,E1 -1165.592,E2 -1165.592} C_VEL
LIN {X 0,Y 594.267,Z 477.957,A -85,B 0,C 180,E1 -1166.61,E2 -1166.61} C_VEL
LIN {X 0,Y 594.226,Z 479.809,A -85,B 0,C 180,E1 -1167.289,E2 -1167.289} C_VEL
LIN {X 0,Y 594.24,Z 481.201,A -85,B 0,C 180,E1 -1167.967,E2 -1167.967} C_VEL
LIN {X 0,Y 594.239,Z 482.784,A -85,B 0,C 180,E1 -1169.323,E2 -1169.323} C_VEL
LIN {X 0,Y 594.236,Z 483,A -85,B 0,C 180,E1 -1170,E2 -1170} C_VEL
LIN {X 0,Y 594.247,Z 482.185,A -85,B 0,C 180,E1 -1171.356,E2 -1171.356} C_VEL
LIN {X 0,Y 594.24,Z 481.201,A -85,B 0,C 180,E1 -1172.034,E2 -1172.034} C_VEL
LIN {X 0,Y 594.226,Z 479.809,A -85,B 0,C 180,E1 -1172.712,E2 -1172.712} C_VEL
LIN {X 0,Y 594.289,Z 476.895,A -85,B 0,C 180,E1 -1173.729,E2 -1173.729} C_VEL
LIN {X 0,Y 594.241,Z 472.949,A -85,B 0,C 180,E1 -1174.749,E2 -1174.749} C_VEL
LIN {X 0,Y 594.304,Z 466.876,A -85,B 0,C 180,E1 -1175.939,E2 -1175.939} C_VEL
LIN {X 0,Y 594.309,Z 460.235,A -85,B 0,C 180,E1 -1176.962,E2 -1176.962} C_VEL
LIN {X 0,Y 594.36,Z 451.988,A -85,B 0,C 180,E1 -1177.987,E2 -1177.987} C_VEL
LIN {X 0,Y 594.405,Z 441.598,A -85,B 0,C 180,E1 -1179.013,E2 -1179.013} C_VEL
LIN {X 0,Y 594.444,Z 430.745,A -85,B 0,C 180,E1 -1179.871,E2 -1179.871} C_VEL
LIN {X 0,Y 594.508,Z 419.775,A -85,B 0,C 180,E1 -1180.558,E2 -1180.558} C_VEL
LIN {X 0,Y 594.602,Z 407.158,A -85,B 0,C 180,E1 -1181.175,E2 -1181.175} C_VEL
LIN {X 0,Y 594.622,Z 395.869,A -85,B 0,C 180,E1 -1181.591,E2 -1181.591} C_VEL
LIN {X 0,Y 594.661,Z 383.5,A -85,B 0,C 180,E1 -1181.915,E2 -1181.915} C_VEL
LIN {X 0,Y 594.696,Z 367.718,A -85,B 0,C 180,E1 -1182.152,E2 -1182.152} C_VEL
LIN {X 0,Y 594.631,Z 272.917,A -85,B 0,C 180,E1 -1183.303,E2 -1183.303} C_VEL
LIN {X 0,Y 594.425,Z 271.001,A -85,B 0,C 180,E1 -1183.373,E2 -1183.373} C_VEL
LIN {X 0,Y 594.49,Z 251.915,A -85,B 0,C 180,E1 -1186.13,E2 -1186.13} C_VEL
LIN {X 0,Y 594.596,Z 233.252,A -85,B 0,C 180,E1 -1188.873,E2 -1188.873} C_VEL
LIN {X 0,Y 594.699,Z 215.717,A -85,B 0,C 180,E1 -1191.491,E2 -1191.491} C_VEL
LIN {X 0,Y 594.382,Z 212.997,A -85,B 0,C 180,E1 -1191.959,E2 -1191.959} C_VEL
LIN {X 0,Y 594.372,Z 212.942,A -85,B 0,C 180,E1 -1194.447,E2 -1194.447} C_VEL
LIN {X 0,Y 594.386,Z 212.939,A -85,B 0,C 180,E1 -1196.7,E2 -1196.7} C_VEL
LIN {X 0,Y 594.38,Z 212.94,A -85,B 0,C 180,E1 -1198.999,E2 -1198.999} C_VEL
LIN {X 0,Y 594.381,Z 212.945,A -85,B 0,C 180,E1 -1201.642,E2 -1201.642} C_VEL
LIN {X 0,Y 594.373,Z 212.943,A -85,B 0,C 180,E1 -1204.58,E2 -1204.58} C_VEL
LIN {X 0,Y 594.394,Z 212.94,A -85,B 0,C 180,E1 -1207.607,E2 -1207.607} C_VEL
LIN {X 0,Y 594.365,Z 212.948,A -85,B 0,C 180,E1 -1210.567,E2 -1210.567} C_VEL
LIN {X 0,Y 594.357,Z 212.942,A -85,B 0,C 180,E1 -1213.3,E2 -1213.3} C_VEL
LIN {X 0,Y 594.368,Z 212.946,A -85,B 0,C 180,E1 -1216.161,E2 -1216.161} C_VEL
LIN {X 0,Y 594.384,Z 212.949,A -85,B 0,C 180,E1 -1218.535,E2 -1218.535} C_VEL
LIN {X 0,Y 594.374,Z 212.942,A -85,B 0,C 180,E1 -1221.297,E2 -1221.297} C_VEL
LIN {X 0,Y 594.353,Z 212.943,A -85,B 0,C 180,E1 -1223.754,E2 -1223.754} C_VEL
LIN {X 0,Y 594.369,Z 212.943,A -85,B 0,C 180,E1 -1226.236,E2 -1226.236} C_VEL
LIN {X 0,Y 594.372,Z 212.946,A -85,B 0,C 180,E1 -1228.648,E2 -1228.648} C_VEL
LIN {X 0,Y 594.383,Z 212.95,A -85,B 0,C 180,E1 -1231.042,E2 -1231.042} C_VEL
LIN {X 0,Y 594.383,Z 212.947,A -85,B 0,C 180,E1 -1233.298,E2 -1233.298} C_VEL
LIN {X 0,Y 594.347,Z 212.947,A -85,B 0,C 180,E1 -1235.575,E2 -1235.575} C_VEL
LIN {X 0,Y 594.361,Z 212.942,A -85,B 0,C 180,E1 -1238.494,E2 -1238.494} C_VEL
LIN {X 0,Y 594.378,Z 212.951,A -85,B 0,C 180,E1 -1241.38,E2 -1241.38} C_VEL
LIN {X 0,Y 594.355,Z 212.943,A -85,B 0,C 180,E1 -1244.216,E2 -1244.216} C_VEL
LIN {X 0,Y 594.359,Z 212.943,A -85,B 0,C 180,E1 -1246.318,E2 -1246.318} C_VEL
LIN {X 0,Y 594.382,Z 212.941,A -85,B 0,C 180,E1 -1249.092,E2 -1249.092} C_VEL
LIN {X 0,Y 594.362,Z 212.952,A -85,B 0,C 180,E1 -1251.84,E2 -1251.84} C_VEL
LIN {X 0,Y 594.353,Z 212.953,A -85,B 0,C 180,E1 -1253.888,E2 -1253.888} C_VEL
LIN {X 0,Y 594.357,Z 212.954,A -85,B 0,C 180,E1 -1255.929,E2 -1255.929} C_VEL
LIN {X 0,Y 594.401,Z 212.948,A -85,B 0,C 180,E1 -1257.964,E2 -1257.964} C_VEL
LIN {X 0,Y 594.396,Z 212.939,A -85,B 0,C 180,E1 -1260.674,E2 -1260.674} C_VEL
LIN {X 0,Y 594.363,Z 212.941,A -85,B 0,C 180,E1 -1263.386,E2 -1263.386} C_VEL
LIN {X 0,Y 594.379,Z 212.948,A -85,B 0,C 180,E1 -1266.105,E2 -1266.105} C_VEL
LIN {X 0,Y 594.364,Z 212.945,A -85,B 0,C 180,E1 -1268.839,E2 -1268.839} C_VEL
LIN {X 0,Y 594.37,Z 212.94,A -85,B 0,C 180,E1 -1271.593,E2 -1271.593} C_VEL
LIN {X 0,Y 594.381,Z 212.947,A -85,B 0,C 180,E1 -1274.373,E2 -1274.373} C_VEL
LIN {X 0,Y 594.345,Z 212.944,A -85,B 0,C 180,E1 -1275.31,E2 -1275.31} C_VEL
LIN {X 0,Y 593.668,Z 213.03,A -85,B 0,C 180,E1 -1275.875,E2 -1275.875} C_VEL
LIN {X 0,Y 590.801,Z 213.394,A -85,B 0,C 180,E1 -1276.793,E2 -1276.793} C_VEL
LIN {X 0,Y 588.392,Z 213.69,A -85,B 0,C 180,E1 -1277.532,E2 -1277.532} C_VEL
LIN {X 0,Y 587.372,Z 213.815,A -85,B 0,C 180,E1 -1278.102,E2 -1278.102} C_VEL
LIN {X 0,Y 587.296,Z 213.825,A -85,B 0,C 180,E1 -1278.295,E2 -1278.295} C_VEL
LIN {X 0,Y 587.345,Z 213.822,A -85,B 0,C 180,E1 -1281.041,E2 -1281.041} C_VEL
LIN {X 0,Y 587.306,Z 213.825,A -85,B 0,C 180,E1 -1283.255,E2 -1283.255} C_VEL
LIN {X 0,Y 587.31,Z 213.821,A -85,B 0,C 180,E1 -1285.513,E2 -1285.513} C_VEL
LIN {X 0,Y 587.329,Z 213.818,A -85,B 0,C 180,E1 -1287.814,E2 -1287.814} C_VEL
LIN {X 0,Y 587.312,Z 213.821,A -85,B 0,C 180,E1 -1290.506,E2 -1290.506} C_VEL
LIN {X 0,Y 587.315,Z 213.829,A -85,B 0,C 180,E1 -1293.108,E2 -1293.108} C_VEL
LIN {X 0,Y 587.319,Z 213.821,A -85,B 0,C 180,E1 -1295.892,E2 -1295.892} C_VEL
LIN {X 0,Y 587.305,Z 213.82,A -85,B 0,C 180,E1 -1298.475,E2 -1298.475} C_VEL
LIN {X 0,Y 587.334,Z 213.822,A -85,B 0,C 180,E1 -1301.151,E2 -1301.151} C_VEL
LIN {X 0,Y 587.301,Z 213.825,A -85,B 0,C 180,E1 -1304.111,E2 -1304.111} C_VEL
LIN {X 0,Y 587.301,Z 213.823,A -85,B 0,C 180,E1 -1306.992,E2 -1306.992} C_VEL
LIN {X 0,Y 587.321,Z 213.83,A -85,B 0,C 180,E1 -1309.974,E2 -1309.974} C_VEL
LIN {X 0,Y 587.377,Z 214,A -85,B 0,C 180,E1 -1311.565,E2 -1311.565} C_VEL
LIN {X 0,Y 587.585,Z 220.263,A -85,B 0,C 180,E1 -1312.626,E2 -1312.626} C_VEL
LIN {X 0,Y 587.462,Z 238.631,A -85,B 0,C 180,E1 -1315.627,E2 -1315.627} C_VEL
LIN {X 0,Y 587.339,Z 256.07,A -85,B 0,C 180,E1 -1318.432,E2 -1318.432} C_VEL
LIN {X 0,Y 587.403,Z 257.363,A -85,B 0,C 180,E1 -1318.559,E2 -1318.559} C_VEL
LIN {X 0,Y 587.851,Z 261.98,A -85,B 0,C 180,E1 -1318.635,E2 -1318.635} C_VEL
LIN {X 0,Y 587.747,Z 364.059,A -85,B 0,C 180,E1 -1319.903,E2 -1319.903} C_VEL
LIN {X 0,Y 587.669,Z 377.706,A -85,B 0,C 180,E1 -1320.22,E2 -1320.22} C_VEL
LIN {X 0,Y 587.639,Z 389.78,A -85,B 0,C 180,E1 -1320.636,E2 -1320.636} C_VEL
LIN {X 0,Y 587.527,Z 400.897,A -85,B 0,C 180,E1 -1321.147,E2 -1321.147} C_VEL
LIN {X 0,Y 587.462,Z 411.995,A -85,B 0,C 180,E1 -1321.8,E2 -1321.8} C_VEL
LIN {X 0,Y 587.403,Z 422.487,A -85,B 0,C 180,E1 -1322.572,E2 -1322.572} C_VEL
LIN {X 0,Y 587.328,Z 431.021,A -85,B 0,C 180,E1 -1323.338,E2 -1323.338} C_VEL
LIN {X 0,Y 587.27,Z 439.812,A -85,B 0,C 180,E1 -1324.29,E2 -1324.29} C_VEL
LIN {X 0,Y 587.248,Z 446.92,A -85,B 0,C 180,E1 -1325.237,E2 -1325.237} C_VEL
LIN {X 0,Y 587.186,Z 453.688,A -85,B 0,C 180,E1 -1326.362,E2 -1326.362} C_VEL
LIN {X 0,Y 587.163,Z 458.942,A -85,B 0,C 180,E1 -1327.479,E2 -1327.479} C_VEL
LIN {X 0,Y 587.163,Z 462.878,A -85,B 0,C 180,E1 -1328.588,E2 -1328.588} C_VEL
LIN {X 0,Y 587.154,Z 465.635,A -85,B 0,C 180,E1 -1329.689,E2 -1329.689} C_VEL
LIN {X 0,Y 587.154,Z 467.535,A -85,B 0,C 180,E1 -1330.997,E2 -1330.997} C_VEL
LIN {X 0,Y 587.128,Z 467.966,A -85,B 0,C 180,E1 -1331.867,E2 -1331.867} C_VEL
LIN {X 0,Y 587.124,Z 467.876,A -85,B 0,C 180,E1 -1332.587,E2 -1332.587} C_VEL
LIN {X 0,Y 587.134,Z 467.312,A -85,B 0,C 180,E1 -1333.305,E2 -1333.305} C_VEL
LIN {X 0,Y 587.149,Z 466.336,A -85,B 0,C 180,E1 -1334.02,E2 -1334.02} C_VEL
LIN {X 0,Y 587.155,Z 464.939,A -85,B 0,C 180,E1 -1334.732,E2 -1334.732} C_VEL
LIN {X 0,Y 587.179,Z 461.992,A -85,B 0,C 180,E1 -1335.789,E2 -1335.789} C_VEL
LIN {X 0,Y 587.186,Z 457.932,A -85,B 0,C 180,E1 -1336.855,E2 -1336.855} C_VEL
LIN {X 0,Y 587.207,Z 451.709,A -85,B 0,C 180,E1 -1338.085,E2 -1338.085} C_VEL
LIN {X 0,Y 587.243,Z 444.924,A -85,B 0,C 180,E1 -1339.135,E2 -1339.135} C_VEL
LIN {X 0,Y 587.305,Z 436.524,A -85,B 0,C 180,E1 -1340.182,E2 -1340.182} C_VEL
LIN {X 0,Y 587.39,Z 425.948,A -85,B 0,C 180,E1 -1341.225,E2 -1341.225} C_VEL
LIN {X 0,Y 587.445,Z 416.152,A -85,B 0,C 180,E1 -1342.005,E2 -1342.005} C_VEL
LIN {X 0,Y 587.491,Z 405.371,A -85,B 0,C 180,E1 -1342.698,E2 -1342.698} C_VEL
LIN {X 0,Y 587.592,Z 392.942,A -85,B 0,C 180,E1 -1343.321,E2 -1343.321} C_VEL
LIN {X 0,Y 587.667,Z 381.375,A -85,B 0,C 180,E1 -1343.759,E2 -1343.759} C_VEL
LIN {X 0,Y 587.721,Z 368.562,A -85,B 0,C 180,E1 -1344.101,E2 -1344.101} C_VEL
LIN {X 0,Y 587.725,Z 353.151,A -85,B 0,C 180,E1 -1344.338,E2 -1344.338} C_VEL
LIN {X 0,Y 587.747,Z 259.433,A -85,B 0,C 180,E1 -1345.488,E2 -1345.488} C_VEL
LIN {X 0,Y 587.369,Z 256.831,A -85,B 0,C 180,E1 -1345.561,E2 -1345.561} C_VEL
LIN {X 0,Y 587.422,Z 240.791,A -85,B 0,C 180,E1 -1348.114,E2 -1348.114} C_VEL
LIN {X 0,Y 587.535,Z 223.96,A -85,B 0,C 180,E1 -1350.857,E2 -1350.857} C_VEL
LIN {X 0,Y 587.493,Z 214.626,A -85,B 0,C 180,E1 -1352.399,E2 -1352.399} C_VEL
LIN {X 0,Y 587.36,Z 213.891,A -85,B 0,C 180,E1 -1352.572,E2 -1352.572} C_VEL
LIN {X 0,Y 587.363,Z 213.815,A -85,B 0,C 180,E1 -1355.493,E2 -1355.493} C_VEL
LIN {X 0,Y 587.346,Z 213.824,A -85,B 0,C 180,E1 -1358.255,E2 -1358.255} C_VEL
LIN {X 0,Y 587.376,Z 213.814,A -85,B 0,C 180,E1 -1361.176,E2 -1361.176} C_VEL
LIN {X 0,Y 587.345,Z 213.82,A -85,B 0,C 180,E1 -1364.275,E2 -1364.275} C_VEL
LIN {X 0,Y 587.339,Z 213.827,A -85,B 0,C 180,E1 -1366.83,E2 -1366.83} C_VEL
LIN {X 0,Y 587.317,Z 213.819,A -85,B 0,C 180,E1 -1369.576,E2 -1369.576} C_VEL
LIN {X 0,Y 587.33,Z 213.818,A -85,B 0,C 180,E1 -1371.774,E2 -1371.774} C_VEL
LIN {X 0,Y 587.333,Z 213.82,A -85,B 0,C 180,E1 -1374.589,E2 -1374.589} C_VEL
LIN {X 0,Y 587.315,Z 213.826,A -85,B 0,C 180,E1 -1377.047,E2 -1377.047} C_VEL
LIN {X 0,Y 587.335,Z 213.826,A -85,B 0,C 180,E1 -1379.38,E2 -1379.38} C_VEL
LIN {X 0,Y 587.332,Z 213.821,A -85,B 0,C 180,E1 -1381.844,E2 -1381.844} C_VEL
LIN {X 0,Y 587.333,Z 213.817,A -85,B 0,C 180,E1 -1384.355,E2 -1384.355} C_VEL
LIN {X 0,Y 587.315,Z 213.819,A -85,B 0,C 180,E1 -1386.749,E2 -1386.749} C_VEL
LIN {X 0,Y 587.326,Z 213.824,A -85,B 0,C 180,E1 -1389.36,E2 -1389.36} C_VEL
LIN {X 0,Y 587.327,Z 213.822,A -85,B 0,C 180,E1 -1392.114,E2 -1392.114} C_VEL
LIN {X 0,Y 587.312,Z 213.82,A -85,B 0,C 180,E1 -1395.095,E2 -1395.095} C_VEL
LIN {X 0,Y 587.317,Z 213.829,A -85,B 0,C 180,E1 -1397.931,E2 -1397.931} C_VEL
LIN {X 0,Y 587.329,Z 213.818,A -85,B 0,C 180,E1 -1400.646,E2 -1400.646} C_VEL
LIN {X 0,Y 587.328,Z 213.817,A -85,B 0,C 180,E1 -1403.294,E2 -1403.294} C_VEL
LIN {X 0,Y 587.354,Z 213.817,A -85,B 0,C 180,E1 -1405.785,E2 -1405.785} C_VEL
LIN {X 0,Y 587.335,Z 213.825,A -85,B 0,C 180,E1 -1408.236,E2 -1408.236} C_VEL
LIN {X 0,Y 587.338,Z 213.819,A -85,B 0,C 180,E1 -1410.868,E2 -1410.868} C_VEL
LIN {X 0,Y 587.344,Z 213.814,A -85,B 0,C 180,E1 -1413.821,E2 -1413.821} C_VEL
LIN {X 0,Y 587.35,Z 213.826,A -85,B 0,C 180,E1 -1416.747,E2 -1416.747} C_VEL
LIN {X 0,Y 587.322,Z 213.819,A -85,B 0,C 180,E1 -1419.699,E2 -1419.699} C_VEL
LIN {X 0,Y 587.345,Z 213.819,A -85,B 0,C 180,E1 -1422.598,E2 -1422.598} C_VEL
LIN {X 0,Y 587.353,Z 213.814,A -85,B 0,C 180,E1 -1425.743,E2 -1425.743} C_VEL
LIN {X 0,Y 587.353,Z 213.818,A -85,B 0,C 180,E1 -1428.862,E2 -1428.862} C_VEL
LIN {X 0,Y 587.367,Z 213.817,A -85,B 0,C 180,E1 -1431.748,E2 -1431.748} C_VEL
LIN {X 0,Y 587.352,Z 213.814,A -85,B 0,C 180,E1 -1434.51,E2 -1434.51} C_VEL
LIN {X 0,Y 587.369,Z 213.816,A -85,B 0,C 180,E1 -1437.26,E2 -1437.26} C_VEL
LIN {X 0,Y 587.38,Z 213.816,A -85,B 0,C 180,E1 -1440.003,E2 -1440.003} C_VEL
LIN {X 0,Y 587.375,Z 213.812,A -85,B 0,C 180,E1 -1442.746,E2 -1442.746} C_VEL
LIN {X 0,Y 587.349,Z 213.819,A -85,B 0,C 180,E1 -1445.496,E2 -1445.496} C_VEL
LIN {X 0,Y 587.365,Z 213.818,A -85,B 0,C 180,E1 -1448.258,E2 -1448.258} C_VEL
LIN {X 0,Y 587.35,Z 213.813,A -85,B 0,C 180,E1 -1451.136,E2 -1451.136} C_VEL
LIN {X 0,Y 587.367,Z 213.824,A -85,B 0,C 180,E1 -1454.262,E2 -1454.262} C_VEL
LIN {X 0,Y 587.349,Z 213.815,A -85,B 0,C 180,E1 -1457.408,E2 -1457.408} C_VEL
LIN {X 0,Y 587.331,Z 213.824,A -85,B 0,C 180,E1 -1460.307,E2 -1460.307} C_VEL
LIN {X 0,Y 587.314,Z 213.821,A -85,B 0,C 180,E1 -1463.261,E2 -1463.261} C_VEL
LIN {X 0,Y 587.333,Z 213.818,A -85,B 0,C 180,E1 -1465.519,E2 -1465.519} C_VEL
LIN {X 0,Y 587.343,Z 213.816,A -85,B 0,C 180,E1 -1467.82,E2 -1467.82} C_VEL
LIN {X 0,Y 587.326,Z 213.821,A -85,B 0,C 180,E1 -1470.509,E2 -1470.509} C_VEL
LIN {X 0,Y 587.339,Z 213.826,A -85,B 0,C 180,E1 -1473.113,E2 -1473.113} C_VEL
LIN {X 0,Y 587.294,Z 213.822,A -85,B 0,C 180,E1 -1475.902,E2 -1475.902} C_VEL
LIN {X 0,Y 587.325,Z 213.819,A -85,B 0,C 180,E1 -1478.482,E2 -1478.482} C_VEL
LIN {X 0,Y 587.34,Z 213.825,A -85,B 0,C 180,E1 -1481.158,E2 -1481.158} C_VEL
LIN {X 0,Y 587.317,Z 213.818,A -85,B 0,C 180,E1 -1484.113,E2 -1484.113} C_VEL
LIN {X 0,Y 587.308,Z 213.821,A -85,B 0,C 180,E1 -1486.994,E2 -1486.994} C_VEL
LIN {X 0,Y 587.313,Z 213.829,A -85,B 0,C 180,E1 -1489.746,E2 -1489.746} C_VEL
LIN {X 0,Y 587.347,Z 213.817,A -85,B 0,C 180,E1 -1492.393,E2 -1492.393} C_VEL
LIN {X 0,Y 587.359,Z 213.824,A -85,B 0,C 180,E1 -1495.78,E2 -1495.78} C_VEL
LIN {X 0,Y 587.341,Z 213.823,A -85,B 0,C 180,E1 -1498.232,E2 -1498.232} C_VEL
LIN {X 0,Y 587.348,Z 213.816,A -85,B 0,C 180,E1 -1500.869,E2 -1500.869} C_VEL
LIN {X 0,Y 587.335,Z 213.821,A -85,B 0,C 180,E1 -1503.722,E2 -1503.722} C_VEL
LIN {X 0,Y 587.311,Z 213.827,A -85,B 0,C 180,E1 -1505.993,E2 -1505.993} C_VEL
LIN {X 0,Y 587.359,Z 214.031,A -85,B 0,C 180,E1 -1507.95,E2 -1507.95} C_VEL
LIN {X 0,Y 587.75,Z 218.358,A -85,B 0,C 180,E1 -1508.645,E2 -1508.645} C_VEL
LIN {X 0,Y 587.588,Z 237.439,A -85,B 0,C 180,E1 -1511.521,E2 -1511.521} C_VEL
LIN {X 0,Y 587.477,Z 255.539,A -85,B 0,C 180,E1 -1514.208,E2 -1514.208} C_VEL
LIN {X 0,Y 587.406,Z 271.274,A -85,B 0,C 180,E1 -1516.486,E2 -1516.486} C_VEL
LIN {X 0,Y 587.867,Z 274.744,A -85,B 0,C 180,E1 -1516.563,E2 -1516.563} C_VEL
LIN {X 0,Y 587.753,Z 378.962,A -85,B 0,C 180,E1 -1517.856,E2 -1517.856} C_VEL
LIN {X 0,Y 587.685,Z 392.229,A -85,B 0,C 180,E1 -1518.161,E2 -1518.161} C_VEL
LIN {X 0,Y 587.603,Z 404.786,A -85,B 0,C 180,E1 -1518.591,E2 -1518.591} C_VEL
LIN {X 0,Y 587.561,Z 416.635,A -85,B 0,C 180,E1 -1519.141,E2 -1519.141} C_VEL
LIN {X 0,Y 587.437,Z 428.207,A -85,B 0,C 180,E1 -1519.836,E2 -1519.836} C_VEL
LIN {X 0,Y 587.392,Z 438.602,A -85,B 0,C 180,E1 -1520.618,E2 -1520.618} C_VEL
LIN {X 0,Y 587.299,Z 447.049,A -85,B 0,C 180,E1 -1521.398,E2 -1521.398} C_VEL
LIN {X 0,Y 587.274,Z 454.963,A -85,B 0,C 180,E1 -1522.263,E2 -1522.263} C_VEL
LIN {X 0,Y 587.231,Z 461.471,A -85,B 0,C 180,E1 -1523.127,E2 -1523.127} C_VEL
LIN {X 0,Y 587.236,Z 467.868,A -85,B 0,C 180,E1 -1524.162,E2 -1524.162} C_VEL
LIN {X 0,Y 587.147,Z 472.951,A -85,B 0,C 180,E1 -1525.194,E2 -1525.194} C_VEL
LIN {X 0,Y 587.213,Z 476.896,A -85,B 0,C 180,E1 -1526.226,E2 -1526.226} C_VEL
LIN {X 0,Y 587.132,Z 479.809,A -85,B 0,C 180,E1 -1527.256,E2 -1527.256} C_VEL
LIN {X 0,Y 587.139,Z 481.2,A -85,B 0,C 180,E1 -1527.942,E2 -1527.942} C_VEL
LIN {X 0,Y 587.14,Z 482.785,A -85,B 0,C 180,E1 -1529.314,E2 -1529.314} C_VEL
LIN {X 0,Y 587.137,Z 483,A -85,B 0,C 180,E1 -1530,E2 -1530} C_VEL
LIN {X 0,Y 587.147,Z 482.185,A -85,B 0,C 180,E1 -1531.372,E2 -1531.372} C_VEL
LIN {X 0,Y 587.139,Z 481.2,A -85,B 0,C 180,E1 -1532.058,E2 -1532.058} C_VEL
LIN {X 0,Y 587.132,Z 479.809,A -85,B 0,C 180,E1 -1532.745,E2 -1532.745} C_VEL
LIN {X 0,Y 587.213,Z 476.895,A -85,B 0,C 180,E1 -1533.775,E2 -1533.775} C_VEL
LIN {X 0,Y 587.147,Z 472.948,A -85,B 0,C 180,E1 -1534.807,E2 -1534.807} C_VEL
LIN {X 0,Y 587.217,Z 466.876,A -85,B 0,C 180,E1 -1536.011,E2 -1536.011} C_VEL
LIN {X 0,Y 587.246,Z 460.236,A -85,B 0,C 180,E1 -1537.046,E2 -1537.046} C_VEL
LIN {X 0,Y 587.298,Z 451.988,A -85,B 0,C 180,E1 -1538.083,E2 -1538.083} C_VEL
LIN {X 0,Y 587.357,Z 441.599,A -85,B 0,C 180,E1 -1539.122,E2 -1539.122} C_VEL
LIN {X 0,Y 587.44,Z 430.744,A -85,B 0,C 180,E1 -1539.99,E2 -1539.99} C_VEL
LIN {X 0,Y 587.525,Z 419.777,A -85,B 0,C 180,E1 -1540.685,E2 -1540.685} C_VEL
LIN {X 0,Y 587.619,Z 408.197,A -85,B 0,C 180,E1 -1541.264,E2 -1541.264} C_VEL
LIN {X 0,Y 587.687,Z 395.867,A -85,B 0,C 180,E1 -1541.73,E2 -1541.73} C_VEL
LIN {X 0,Y 587.715,Z 383.498,A -85,B 0,C 180,E1 -1542.058,E2 -1542.058} C_VEL
LIN {X 0,Y 587.769,Z 367.718,A -85,B 0,C 180,E1 -1542.298,E2 -1542.298} C_VEL
LIN {X 0,Y 587.754,Z 273.589,A -85,B 0,C 180,E1 -1543.454,E2 -1543.454} C_VEL
LIN {X 0,Y 587.406,Z 271.268,A -85,B 0,C 180,E1 -1543.514,E2 -1543.514} C_VEL
LIN {X 0,Y 587.484,Z 253.122,A -85,B 0,C 180,E1 -1546.149,E2 -1546.149} C_VEL
LIN {X 0,Y 587.609,Z 235.023,A -85,B 0,C 180,E1 -1548.84,E2 -1548.84} C_VEL
LIN {X 0,Y 587.763,Z 216.92,A -85,B 0,C 180,E1 -1551.574,E2 -1551.574} C_VEL
LIN {X 0,Y 587.346,Z 213.897,A -85,B 0,C 180,E1 -1552.097,E2 -1552.097} C_VEL
LIN {X 0,Y 587.32,Z 213.821,A -85,B 0,C 180,E1 -1554.76,E2 -1554.76} C_VEL
LIN {X 0,Y 587.348,Z 213.825,A -85,B 0,C 180,E1 -1557.69,E2 -1557.69} C_VEL
LIN {X 0,Y 587.329,Z 213.82,A -85,B 0,C 180,E1 -1560.507,E2 -1560.507} C_VEL
LIN {X 0,Y 587.34,Z 213.818,A -85,B 0,C 180,E1 -1563.396,E2 -1563.396} C_VEL
LIN {X 0,Y 587.287,Z 213.83,A -85,B 0,C 180,E1 -1565.9,E2 -1565.9} C_VEL
LIN {X 0,Y 587.325,Z 213.824,A -85,B 0,C 180,E1 -1568.48,E2 -1568.48} C_VEL
LIN {X 0,Y 587.338,Z 213.817,A -85,B 0,C 180,E1 -1571.157,E2 -1571.157} C_VEL
LIN {X 0,Y 587.311,Z 213.825,A -85,B 0,C 180,E1 -1574.11,E2 -1574.11} C_VEL
LIN {X 0,Y 587.302,Z 213.823,A -85,B 0,C 180,E1 -1576.991,E2 -1576.991} C_VEL
LIN {X 0,Y 587.314,Z 213.82,A -85,B 0,C 180,E1 -1579.744,E2 -1579.744} C_VEL
LIN {X 0,Y 587.349,Z 213.821,A -85,B 0,C 180,E1 -1582.391,E2 -1582.391} C_VEL
LIN {X 0,Y 587.34,Z 213.817,A -85,B 0,C 180,E1 -1585.654,E2 -1585.654} C_VEL
LIN {X 0,Y 587.34,Z 213.817,A -85,B 0,C 180,E1 -1588.229,E2 -1588.229} C_VEL
LIN {X 0,Y 587.35,Z 213.824,A -85,B 0,C 180,E1 -1590.867,E2 -1590.867} C_VEL
LIN {X 0,Y 587.313,Z 213.821,A -85,B 0,C 180,E1 -1593.828,E2 -1593.828} C_VEL
LIN {X 0,Y 587.31,Z 213.823,A -85,B 0,C 180,E1 -1596.739,E2 -1596.739} C_VEL
LIN {X 0,Y 587.325,Z 213.822,A -85,B 0,C 180,E1 -1599.693,E2 -1599.693} C_VEL
LIN {X 0,Y 587.297,Z 213.825,A -85,B 0,C 180,E1 -1601.87,E2 -1601.87} C_VEL
LIN {X 0,Y 587.315,Z 213.821,A -85,B 0,C 180,E1 -1604.022,E2 -1604.022} C_VEL
LIN {X 0,Y 587.339,Z 213.818,A -85,B 0,C 180,E1 -1606.151,E2 -1606.151} C_VEL
LIN {X 0,Y 587.348,Z 213.816,A -85,B 0,C 180,E1 -1608.96,E2 -1608.96} C_VEL
LIN {X 0,Y 587.328,Z 213.83,A -85,B 0,C 180,E1 -1611.741,E2 -1611.741} C_VEL
LIN {X 0,Y 587.311,Z 213.831,A -85,B 0,C 180,E1 -1613.815,E2 -1613.815} C_VEL
LIN {X 0,Y 587.312,Z 213.831,A -85,B 0,C 180,E1 -1615.88,E2 -1615.88} C_VEL
LIN {X 0,Y 587.371,Z 213.824,A -85,B 0,C 180,E1 -1617.94,E2 -1617.94} C_VEL
LIN {X 0,Y 587.369,Z 213.815,A -85,B 0,C 180,E1 -1620.682,E2 -1620.682} C_VEL
LIN {X 0,Y 587.316,Z 213.819,A -85,B 0,C 180,E1 -1623.427,E2 -1623.427} C_VEL
LIN {X 0,Y 587.33,Z 213.828,A -85,B 0,C 180,E1 -1626.179,E2 -1626.179} C_VEL
LIN {X 0,Y 587.311,Z 213.822,A -85,B 0,C 180,E1 -1628.946,E2 -1628.946} C_VEL
LIN {X 0,Y 587.321,Z 213.819,A -85,B 0,C 180,E1 -1631.734,E2 -1631.734} C_VEL
LIN {X 0,Y 587.329,Z 213.829,A -85,B 0,C 180,E1 -1634.55,E2 -1634.55} C_VEL
LIN {X 0,Y 587.334,Z 213.818,A -85,B 0,C 180,E1 -1637.402,E2 -1637.402} C_VEL
LIN {X 0,Y 587.296,Z 213.825,A -85,B 0,C 180,E1 -1638.295,E2 -1638.295} C_VEL
LIN {X 0,Y 586.655,Z 213.911,A -85,B 0,C 180,E1 -1638.867,E2 -1638.867} C_VEL
LIN {X 0,Y 583.832,Z 214.263,A -85,B 0,C 180,E1 -1639.796,E2 -1639.796} C_VEL
LIN {X 0,Y 581.422,Z 214.562,A -85,B 0,C 180,E1 -1640.543,E2 -1640.543} C_VEL
LIN {X 0,Y 580.37,Z 214.69,A -85,B 0,C 180,E1 -1641.119,E2 -1641.119} C_VEL
LIN {X 0,Y 580.276,Z 214.699,A -85,B 0,C 180,E1 -1641.315,E2 -1641.315} C_VEL
LIN {X 0,Y 580.259,Z 214.7,A -85,B 0,C 180,E1 -1643.554,E2 -1643.554} C_VEL
LIN {X 0,Y 580.269,Z 214.696,A -85,B 0,C 180,E1 -1645.845,E2 -1645.845} C_VEL
LIN {X 0,Y 580.282,Z 214.696,A -85,B 0,C 180,E1 -1648.181,E2 -1648.181} C_VEL
LIN {X 0,Y 580.265,Z 214.701,A -85,B 0,C 180,E1 -1650.691,E2 -1650.691} C_VEL
LIN {X 0,Y 580.279,Z 214.706,A -85,B 0,C 180,E1 -1653.313,E2 -1653.313} C_VEL
LIN {X 0,Y 580.272,Z 214.701,A -85,B 0,C 180,E1 -1655.76,E2 -1655.76} C_VEL
LIN {X 0,Y 580.261,Z 214.699,A -85,B 0,C 180,E1 -1658.142,E2 -1658.142} C_VEL
LIN {X 0,Y 580.288,Z 214.696,A -85,B 0,C 180,E1 -1660.838,E2 -1660.838} C_VEL
LIN {X 0,Y 580.256,Z 214.71,A -85,B 0,C 180,E1 -1663.653,E2 -1663.653} C_VEL
LIN {X 0,Y 580.251,Z 214.7,A -85,B 0,C 180,E1 -1666.605,E2 -1666.605} C_VEL
LIN {X 0,Y 580.291,Z 214.697,A -85,B 0,C 180,E1 -1669.156,E2 -1669.156} C_VEL
LIN {X 0,Y 580.337,Z 214.843,A -85,B 0,C 180,E1 -1671.443,E2 -1671.443} C_VEL
LIN {X 0,Y 580.635,Z 218.566,A -85,B 0,C 180,E1 -1672.1,E2 -1672.1} C_VEL
LIN {X 0,Y 580.486,Z 236.699,A -85,B 0,C 180,E1 -1675.106,E2 -1675.106} C_VEL
LIN {X 0,Y 580.359,Z 254.119,A -85,B 0,C 180,E1 -1677.95,E2 -1677.95} C_VEL
LIN {X 0,Y 580.33,Z 256.862,A -85,B 0,C 180,E1 -1678.363,E2 -1678.363} C_VEL
LIN {X 0,Y 580.955,Z 261.312,A -85,B 0,C 180,E1 -1678.465,E2 -1678.465} C_VEL
LIN {X 0,Y 580.802,Z 364.092,A -85,B 0,C 180,E1 -1679.756,E2 -1679.756} C_VEL
LIN {X 0,Y 580.735,Z 377.751,A -85,B 0,C 180,E1 -1680.078,E2 -1680.078} C_VEL
LIN {X 0,Y 580.67,Z 389.256,A -85,B 0,C 180,E1 -1680.477,E2 -1680.477} C_VEL
LIN {X 0,Y 580.531,Z 401.335,A -85,B 0,C 180,E1 -1681.037,E2 -1681.037} C_VEL
LIN {X 0,Y 580.455,Z 412.715,A -85,B 0,C 180,E1 -1681.724,E2 -1681.724} C_VEL
LIN {X 0,Y 580.361,Z 422.413,A -85,B 0,C 180,E1 -1682.45,E2 -1682.45} C_VEL
LIN {X 0,Y 580.291,Z 430.549,A -85,B 0,C 180,E1 -1683.183,E2 -1683.183} C_VEL
LIN {X 0,Y 580.215,Z 439.405,A -85,B 0,C 180,E1 -1684.147,E2 -1684.147} C_VEL
LIN {X 0,Y 580.182,Z 446.811,A -85,B 0,C 180,E1 -1685.137,E2 -1685.137} C_VEL
LIN {X 0,Y 580.131,Z 452.432,A -85,B 0,C 180,E1 -1686.056,E2 -1686.056} C_VEL
LIN {X 0,Y 580.107,Z 457.988,A -85,B 0,C 180,E1 -1687.19,E2 -1687.19} C_VEL
LIN {X 0,Y 580.076,Z 462.17,A -85,B 0,C 180,E1 -1688.313,E2 -1688.313} C_VEL
LIN {X 0,Y 580.068,Z 465.158,A -85,B 0,C 180,E1 -1689.429,E2 -1689.429} C_VEL
LIN {X 0,Y 580.05,Z 466.531,A -85,B 0,C 180,E1 -1690.168,E2 -1690.168} C_VEL
LIN {X 0,Y 580.062,Z 467.465,A -85,B 0,C 180,E1 -1690.905,E2 -1690.905} C_VEL
LIN {X 0,Y 580.035,Z 467.914,A -85,B 0,C 180,E1 -1691.637,E2 -1691.637} C_VEL
LIN {X 0,Y 580.032,Z 467.934,A -85,B 0,C 180,E1 -1692.367,E2 -1692.367} C_VEL
LIN {X 0,Y 580.055,Z 467.497,A -85,B 0,C 180,E1 -1693.151,E2 -1693.151} C_VEL
LIN {X 0,Y 580.049,Z 466.692,A -85,B 0,C 180,E1 -1693.819,E2 -1693.819} C_VEL
LIN {X 0,Y 580.061,Z 465.406,A -85,B 0,C 180,E1 -1694.541,E2 -1694.541} C_VEL
LIN {X 0,Y 580.09,Z 462.322,A -85,B 0,C 180,E1 -1695.726,E2 -1695.726} C_VEL
LIN {X 0,Y 580.091,Z 458.842,A -85,B 0,C 180,E1 -1696.691,E2 -1696.691} C_VEL
LIN {X 0,Y 580.104,Z 453.888,A -85,B 0,C 180,E1 -1697.759,E2 -1697.759} C_VEL
LIN {X 0,Y 580.177,Z 447.53,A -85,B 0,C 180,E1 -1698.842,E2 -1698.842} C_VEL
LIN {X 0,Y 580.221,Z 439.899,A -85,B 0,C 180,E1 -1699.884,E2 -1699.884} C_VEL
LIN {X 0,Y 580.308,Z 430.197,A -85,B 0,C 180,E1 -1700.941,E2 -1700.941} C_VEL
LIN {X 0,Y 580.386,Z 420.221,A -85,B 0,C 180,E1 -1701.82,E2 -1701.82} C_VEL
LIN {X 0,Y 580.47,Z 408.98,A -85,B 0,C 180,E1 -1702.609,E2 -1702.609} C_VEL
LIN {X 0,Y 580.582,Z 397.115,A -85,B 0,C 180,E1 -1703.266,E2 -1703.266} C_VEL
LIN {X 0,Y 580.679,Z 384.647,A -85,B 0,C 180,E1 -1703.79,E2 -1703.79} C_VEL
LIN {X 0,Y 580.743,Z 371.364,A -85,B 0,C 180,E1 -1704.183,E2 -1704.183} C_VEL
LIN {X 0,Y 580.796,Z 358.298,A -85,B 0,C 180,E1 -1704.423,E2 -1704.423} C_VEL
LIN {X 0,Y 580.859,Z 260.207,A -85,B 0,C 180,E1 -1705.641,E2 -1705.641} C_VEL
LIN {X 0,Y 580.373,Z 256.865,A -85,B 0,C 180,E1 -1705.724,E2 -1705.724} C_VEL
LIN {X 0,Y 580.393,Z 241.091,A -85,B 0,C 180,E1 -1708.265,E2 -1708.265} C_VEL
LIN {X 0,Y 580.575,Z 224.263,A -85,B 0,C 180,E1 -1711.04,E2 -1711.04} C_VEL
LIN {X 0,Y 580.535,Z 215.972,A -85,B 0,C 180,E1 -1712.428,E2 -1712.428} C_VEL
LIN {X 0,Y 580.327,Z 214.765,A -85,B 0,C 180,E1 -1712.69,E2 -1712.69} C_VEL
LIN {X 0,Y 580.326,Z 214.692,A -85,B 0,C 180,E1 -1715.559,E2 -1715.559} C_VEL
LIN {X 0,Y 580.311,Z 214.702,A -85,B 0,C 180,E1 -1718.356,E2 -1718.356} C_VEL
LIN {X 0,Y 580.329,Z 214.691,A -85,B 0,C 180,E1 -1721.234,E2 -1721.234} C_VEL
LIN {X 0,Y 580.316,Z 214.697,A -85,B 0,C 180,E1 -1724.361,E2 -1724.361} C_VEL
LIN {X 0,Y 580.315,Z 214.7,A -85,B 0,C 180,E1 -1726.934,E2 -1726.934} C_VEL
LIN {X 0,Y 580.278,Z 214.694,A -85,B 0,C 180,E1 -1729.823,E2 -1729.823} C_VEL
LIN {X 0,Y 580.293,Z 214.694,A -85,B 0,C 180,E1 -1732.051,E2 -1732.051} C_VEL
LIN {X 0,Y 580.281,Z 214.705,A -85,B 0,C 180,E1 -1735.081,E2 -1735.081} C_VEL
LIN {X 0,Y 580.284,Z 214.694,A -85,B 0,C 180,E1 -1737.868,E2 -1737.868} C_VEL
LIN {X 0,Y 580.276,Z 214.698,A -85,B 0,C 180,E1 -1740.704,E2 -1740.704} C_VEL
LIN {X 0,Y 580.298,Z 214.703,A -85,B 0,C 180,E1 -1743.325,E2 -1743.325} C_VEL
LIN {X 0,Y 580.297,Z 214.7,A -85,B 0,C 180,E1 -1745.772,E2 -1745.772} C_VEL
LIN {X 0,Y 580.272,Z 214.699,A -85,B 0,C 180,E1 -1748.147,E2 -1748.147} C_VEL
LIN {X 0,Y 580.295,Z 214.693,A -85,B 0,C 180,E1 -1750.843,E2 -1750.843} C_VEL
LIN {X 0,Y 580.262,Z 214.704,A -85,B 0,C 180,E1 -1753.659,E2 -1753.659} C_VEL
LIN {X 0,Y 580.266,Z 214.699,A -85,B 0,C 180,E1 -1756.61,E2 -1756.61} C_VEL
LIN {X 0,Y 580.293,Z 214.693,A -85,B 0,C 180,E1 -1759.163,E2 -1759.163} C_VEL
LIN {X 0,Y 580.266,Z 214.702,A -85,B 0,C 180,E1 -1761.929,E2 -1761.929} C_VEL
LIN {X 0,Y 580.293,Z 214.702,A -85,B 0,C 180,E1 -1764.461,E2 -1764.461} C_VEL
LIN {X 0,Y 580.272,Z 214.699,A -85,B 0,C 180,E1 -1766.979,E2 -1766.979} C_VEL
LIN {X 0,Y 580.288,Z 214.694,A -85,B 0,C 180,E1 -1769.43,E2 -1769.43} C_VEL
LIN {X 0,Y 580.299,Z 214.694,A -85,B 0,C 180,E1 -1772.14,E2 -1772.14} C_VEL
LIN {X 0,Y 580.291,Z 214.701,A -85,B 0,C 180,E1 -1774.924,E2 -1774.924} C_VEL
LIN {X 0,Y 580.312,Z 214.696,A -85,B 0,C 180,E1 -1777.203,E2 -1777.203} C_VEL
LIN {X 0,Y 580.294,Z 214.695,A -85,B 0,C 180,E1 -1780.182,E2 -1780.182} C_VEL
LIN {X 0,Y 580.317,Z 214.697,A -85,B 0,C 180,E1 -1783.107,E2 -1783.107} C_VEL
LIN {X 0,Y 580.315,Z 214.689,A -85,B 0,C 180,E1 -1785.987,E2 -1785.987} C_VEL
LIN {X 0,Y 580.323,Z 214.694,A -85,B 0,C 180,E1 -1788.831,E2 -1788.831} C_VEL
LIN {X 0,Y 580.33,Z 214.695,A -85,B 0,C 180,E1 -1791.647,E2 -1791.647} C_VEL
LIN {X 0,Y 580.32,Z 214.69,A -85,B 0,C 180,E1 -1794.444,E2 -1794.444} C_VEL
LIN {X 0,Y 580.335,Z 214.691,A -85,B 0,C 180,E1 -1797.227,E2 -1797.227} C_VEL
LIN {X 0,Y 580.35,Z 214.691,A -85,B 0,C 180,E1 -1800.003,E2 -1800.003} C_VEL
LIN {X 0,Y 580.34,Z 214.688,A -85,B 0,C 180,E1 -1802.78,E2 -1802.78} C_VEL
LIN {X 0,Y 580.317,Z 214.696,A -85,B 0,C 180,E1 -1805.563,E2 -1805.563} C_VEL
LIN {X 0,Y 580.327,Z 214.692,A -85,B 0,C 180,E1 -1808.359,E2 -1808.359} C_VEL
LIN {X 0,Y 580.302,Z 214.69,A -85,B 0,C 180,E1 -1811.194,E2 -1811.194} C_VEL
LIN {X 0,Y 580.325,Z 214.697,A -85,B 0,C 180,E1 -1814.019,E2 -1814.019} C_VEL
LIN {X 0,Y 580.316,Z 214.693,A -85,B 0,C 180,E1 -1816.916,E2 -1816.916} C_VEL
LIN {X 0,Y 580.29,Z 214.695,A -85,B 0,C 180,E1 -1819.825,E2 -1819.825} C_VEL
LIN {X 0,Y 580.272,Z 214.698,A -85,B 0,C 180,E1 -1822.055,E2 -1822.055} C_VEL
LIN {X 0,Y 580.309,Z 214.697,A -85,B 0,C 180,E1 -1825.082,E2 -1825.082} C_VEL
LIN {X 0,Y 580.298,Z 214.695,A -85,B 0,C 180,E1 -1828.188,E2 -1828.188} C_VEL
LIN {X 0,Y 580.277,Z 214.702,A -85,B 0,C 180,E1 -1830.694,E2 -1830.694} C_VEL
LIN {X 0,Y 580.286,Z 214.701,A -85,B 0,C 180,E1 -1833.314,E2 -1833.314} C_VEL
LIN {X 0,Y 580.248,Z 214.701,A -85,B 0,C 180,E1 -1835.757,E2 -1835.757} C_VEL
LIN {X 0,Y 580.29,Z 214.694,A -85,B 0,C 180,E1 -1838.148,E2 -1838.148} C_VEL
LIN {X 0,Y 580.302,Z 214.697,A -85,B 0,C 180,E1 -1840.845,E2 -1840.845} C_VEL
LIN {X 0,Y 580.275,Z 214.7,A -85,B 0,C 180,E1 -1843.66,E2 -1843.66} C_VEL
LIN {X 0,Y 580.248,Z 214.698,A -85,B 0,C 180,E1 -1846.614,E2 -1846.614} C_VEL
LIN {X 0,Y 580.299,Z 214.697,A -85,B 0,C 180,E1 -1849.157,E2 -1849.157} C_VEL
LIN {X 0,Y 580.292,Z 214.702,A -85,B 0,C 180,E1 -1851.928,E2 -1851.928} C_VEL
LIN {X 0,Y 580.253,Z 214.701,A -85,B 0,C 180,E1 -1854.453,E2 -1854.453} C_VEL
LIN {X 0,Y 580.293,Z 214.694,A -85,B 0,C 180,E1 -1856.976,E2 -1856.976} C_VEL
LIN {X 0,Y 580.288,Z 214.697,A -85,B 0,C 180,E1 -1859.425,E2 -1859.425} C_VEL
LIN {X 0,Y 580.3,Z 214.705,A -85,B 0,C 180,E1 -1862.143,E2 -1862.143} C_VEL
LIN {X 0,Y 580.294,Z 214.697,A -85,B 0,C 180,E1 -1864.92,E2 -1864.92} C_VEL
LIN {X 0,Y 580.318,Z 214.898,A -85,B 0,C 180,E1 -1867.809,E2 -1867.809} C_VEL
LIN {X 0,Y 580.804,Z 219.459,A -85,B 0,C 180,E1 -1868.548,E2 -1868.548} C_VEL
LIN {X 0,Y 580.627,Z 238.646,A -85,B 0,C 180,E1 -1871.474,E2 -1871.474} C_VEL
LIN {X 0,Y 580.474,Z 256.745,A -85,B 0,C 180,E1 -1874.192,E2 -1874.192} C_VEL
LIN {X 0,Y 580.385,Z 271.285,A -85,B 0,C 180,E1 -1876.32,E2 -1876.32} C_VEL
LIN {X 0,Y 580.974,Z 276.532,A -85,B 0,C 180,E1 -1876.423,E2 -1876.423} C_VEL
LIN {X 0,Y 580.807,Z 378.961,A -85,B 0,C 180,E1 -1877.708,E2 -1877.708} C_VEL
LIN {X 0,Y 580.744,Z 392.229,A -85,B 0,C 180,E1 -1878.017,E2 -1878.017} C_VEL
LIN {X 0,Y 580.642,Z 405.501,A -85,B 0,C 180,E1 -1878.48,E2 -1878.48} C_VEL
LIN {X 0,Y 580.563,Z 416.633,A -85,B 0,C 180,E1 -1879.009,E2 -1879.009} C_VEL
LIN {X 0,Y 580.418,Z 428.206,A -85,B 0,C 180,E1 -1879.712,E2 -1879.712} C_VEL
LIN {X 0,Y 580.343,Z 438.604,A -85,B 0,C 180,E1 -1880.503,E2 -1880.503} C_VEL
LIN {X 0,Y 580.263,Z 447.064,A -85,B 0,C 180,E1 -1881.292,E2 -1881.292} C_VEL
LIN {X 0,Y 580.222,Z 454.963,A -85,B 0,C 180,E1 -1882.168,E2 -1882.168} C_VEL
LIN {X 0,Y 580.157,Z 462.642,A -85,B 0,C 180,E1 -1883.22,E2 -1883.22} C_VEL
LIN {X 0,Y 580.139,Z 469.681,A -85,B 0,C 180,E1 -1884.439,E2 -1884.439} C_VEL
LIN {X 0,Y 580.108,Z 474.373,A -85,B 0,C 180,E1 -1885.484,E2 -1885.484} C_VEL
LIN {X 0,Y 580.123,Z 477.958,A -85,B 0,C 180,E1 -1886.528,E2 -1886.528} C_VEL
LIN {X 0,Y 580.043,Z 479.809,A -85,B 0,C 180,E1 -1887.222,E2 -1887.222} C_VEL
LIN {X 0,Y 580.038,Z 481.199,A -85,B 0,C 180,E1 -1887.917,E2 -1887.917} C_VEL
LIN {X 0,Y 580.04,Z 482.785,A -85,B 0,C 180,E1 -1889.306,E2 -1889.306} C_VEL
LIN {X 0,Y 580.037,Z 483,A -85,B 0,C 180,E1 -1890,E2 -1890} C_VEL
LIN {X 0,Y 580.046,Z 482.186,A -85,B 0,C 180,E1 -1891.389,E2 -1891.389} C_VEL
LIN {X 0,Y 580.038,Z 481.199,A -85,B 0,C 180,E1 -1892.083,E2 -1892.083} C_VEL
LIN {X 0,Y 580.043,Z 479.809,A -85,B 0,C 180,E1 -1892.778,E2 -1892.778} C_VEL
LIN {X 0,Y 580.11,Z 476.895,A -85,B 0,C 180,E1 -1893.821,E2 -1893.821} C_VEL
LIN {X 0,Y 580.053,Z 472.948,A -85,B 0,C 180,E1 -1894.865,E2 -1894.865} C_VEL
LIN {X 0,Y 580.14,Z 466.876,A -85,B 0,C 180,E1 -1896.085,E2 -1896.085} C_VEL
LIN {X 0,Y 580.186,Z 460.236,A -85,B 0,C 180,E1 -1897.133,E2 -1897.133} C_VEL
LIN {X 0,Y 580.247,Z 451.989,A -85,B 0,C 180,E1 -1898.182,E2 -1898.182} C_VEL
LIN {X 0,Y 580.333,Z 441.6,A -85,B 0,C 180,E1 -1899.234,E2 -1899.234} C_VEL
LIN {X 0,Y 580.434,Z 430.744,A -85,B 0,C 180,E1 -1900.112,E2 -1900.112} C_VEL
LIN {X 0,Y 580.538,Z 419.779,A -85,B 0,C 180,E1 -1900.815,E2 -1900.815} C_VEL
LIN {X 0,Y 580.665,Z 407.549,A -85,B 0,C 180,E1 -1901.429,E2 -1901.429} C_VEL
LIN {X 0,Y 580.734,Z 395.865,A -85,B 0,C 180,E1 -1901.873,E2 -1901.873} C_VEL
LIN {X 0,Y 580.787,Z 383.497,A -85,B 0,C 180,E1 -1902.204,E2 -1902.204} C_VEL
LIN {X 0,Y 580.833,Z 367.718,A -85,B 0,C 180,E1 -1902.447,E2 -1902.447} C_VEL
LIN {X 0,Y 580.904,Z 274.706,A -85,B 0,C 180,E1 -1903.601,E2 -1903.601} C_VEL
LIN {X 0,Y 580.386,Z 271.28,A -85,B 0,C 180,E1 -1903.681,E2 -1903.681} C_VEL
LIN {X 0,Y 580.502,Z 253.122,A -85,B 0,C 180,E1 -1906.349,E2 -1906.349} C_VEL
LIN {X 0,Y 580.649,Z 235.023,A -85,B 0,C 180,E1 -1909.075,E2 -1909.075} C_VEL
LIN {X 0,Y 580.825,Z 218.119,A -85,B 0,C 180,E1 -1911.657,E2 -1911.657} C_VEL
LIN {X 0,Y 580.307,Z 214.774,A -85,B 0,C 180,E1 -1912.239,E2 -1912.239} C_VEL
LIN {X 0,Y 580.295,Z 214.698,A -85,B 0,C 180,E1 -1915.08,E2 -1915.08} C_VEL
LIN {X 0,Y 580.295,Z 214.705,A -85,B 0,C 180,E1 -1917.856,E2 -1917.856} C_VEL
LIN {X 0,Y 580.279,Z 214.697,A -85,B 0,C 180,E1 -1920.692,E2 -1920.692} C_VEL
LIN {X 0,Y 580.309,Z 214.693,A -85,B 0,C 180,E1 -1923.315,E2 -1923.315} C_VEL
LIN {X 0,Y 580.238,Z 214.706,A -85,B 0,C 180,E1 -1925.754,E2 -1925.754} C_VEL
LIN {X 0,Y 580.292,Z 214.705,A -85,B 0,C 180,E1 -1928.146,E2 -1928.146} C_VEL
LIN {X 0,Y 580.3,Z 214.696,A -85,B 0,C 180,E1 -1930.843,E2 -1930.843} C_VEL
LIN {X 0,Y 580.249,Z 214.7,A -85,B 0,C 180,E1 -1933.661,E2 -1933.661} C_VEL
LIN {X 0,Y 580.273,Z 214.704,A -85,B 0,C 180,E1 -1936.61,E2 -1936.61} C_VEL
LIN {X 0,Y 580.302,Z 214.696,A -85,B 0,C 180,E1 -1939.155,E2 -1939.155} C_VEL
LIN {X 0,Y 580.294,Z 214.695,A -85,B 0,C 180,E1 -1941.927,E2 -1941.927} C_VEL
LIN {X 0,Y 580.24,Z 214.706,A -85,B 0,C 180,E1 -1944.45,E2 -1944.45} C_VEL
LIN {X 0,Y 580.292,Z 214.703,A -85,B 0,C 180,E1 -1946.973,E2 -1946.973} C_VEL
LIN {X 0,Y 580.288,Z 214.698,A -85,B 0,C 180,E1 -1949.423,E2 -1949.423} C_VEL
LIN {X 0,Y 580.254,Z 214.699,A -85,B 0,C 180,E1 -1952.15,E2 -1952.15} C_VEL
LIN {X 0,Y 580.289,Z 214.702,A -85,B 0,C 180,E1 -1954.917,E2 -1954.917} C_VEL
LIN {X 0,Y 580.259,Z 214.7,A -85,B 0,C 180,E1 -1957.945,E2 -1957.945} C_VEL
LIN {X 0,Y 580.304,Z 214.696,A -85,B 0,C 180,E1 -1960.911,E2 -1960.911} C_VEL
LIN {X 0,Y 580.273,Z 214.701,A -85,B 0,C 180,E1 -1963.823,E2 -1963.823} C_VEL
LIN {X 0,Y 580.31,Z 214.696,A -85,B 0,C 180,E1 -1965.98,E2 -1965.98} C_VEL
LIN {X 0,Y 580.311,Z 214.692,A -85,B 0,C 180,E1 -1968.824,E2 -1968.824} C_VEL
LIN {X 0,Y 580.301,Z 214.703,A -85,B 0,C 180,E1 -1971.641,E2 -1971.641} C_VEL
LIN {X 0,Y 580.272,Z 214.707,A -85,B 0,C 180,E1 -1973.739,E2 -1973.739} C_VEL
LIN {X 0,Y 580.268,Z 214.707,A -85,B 0,C 180,E1 -1975.83,E2 -1975.83} C_VEL
LIN {X 0,Y 580.341,Z 214.699,A -85,B 0,C 180,E1 -1977.915,E2 -1977.915} C_VEL
LIN {X 0,Y 580.343,Z 214.69,A -85,B 0,C 180,E1 -1980.691,E2 -1980.691} C_VEL
LIN {X 0,Y 580.32,Z 214.691,A -85,B 0,C 180,E1 -1982.773,E2 -1982.773} C_VEL
LIN {X 0,Y 580.314,Z 214.693,A -85,B 0,C 180,E1 -1985.556,E2 -1985.556} C_VEL
LIN {X 0,Y 580.321,Z 214.702,A -85,B 0,C 180,E1 -1988.353,E2 -1988.353} C_VEL
LIN {X 0,Y 580.294,Z 214.694,A -85,B 0,C 180,E1 -1991.187,E2 -1991.187} C_VEL
LIN {X 0,Y 580.314,Z 214.694,A -85,B 0,C 180,E1 -1994.013,E2 -1994.013} C_VEL
LIN {X 0,Y 580.302,Z 214.7,A -85,B 0,C 180,E1 -1996.91,E2 -1996.91} C_VEL
LIN {X 0,Y 580.276,Z 214.696,A -85,B 0,C 180,E1 -1999.819,E2 -1999.819} C_VEL
LIN {X 0,Y 580.276,Z 214.699,A -85,B 0,C 180,E1 -2001.315,E2 -2001.315} C_VEL
LIN {X 0,Y 579.579,Z 214.786,A -85,B 0,C 180,E1 -2001.894,E2 -2001.894} C_VEL
LIN {X 0,Y 576.698,Z 215.153,A -85,B 0,C 180,E1 -2002.834,E2 -2002.834} C_VEL
LIN {X 0,Y 574.298,Z 215.446,A -85,B 0,C 180,E1 -2003.59,E2 -2003.59} C_VEL
LIN {X 0,Y 573.297,Z 215.567,A -85,B 0,C 180,E1 -2004.174,E2 -2004.174} C_VEL
LIN {X 0,Y 573.23,Z 215.577,A -85,B 0,C 180,E1 -2004.372,E2 -2004.372} C_VEL
LIN {X 0,Y 573.233,Z 215.582,A -85,B 0,C 180,E1 -2006.972,E2 -2006.972} C_VEL
LIN {X 0,Y 573.222,Z 215.579,A -85,B 0,C 180,E1 -2009.484,E2 -2009.484} C_VEL
LIN {X 0,Y 573.232,Z 215.574,A -85,B 0,C 180,E1 -2012.225,E2 -2012.225} C_VEL
LIN {X 0,Y 573.229,Z 215.577,A -85,B 0,C 180,E1 -2014.77,E2 -2014.77} C_VEL
LIN {X 0,Y 573.227,Z 215.582,A -85,B 0,C 180,E1 -2017.162,E2 -2017.162} C_VEL
LIN {X 0,Y 573.221,Z 215.584,A -85,B 0,C 180,E1 -2019.603,E2 -2019.603} C_VEL
LIN {X 0,Y 573.209,Z 215.578,A -85,B 0,C 180,E1 -2022.396,E2 -2022.396} C_VEL
LIN {X 0,Y 573.193,Z 215.58,A -85,B 0,C 180,E1 -2024.672,E2 -2024.672} C_VEL
LIN {X 0,Y 573.229,Z 215.584,A -85,B 0,C 180,E1 -2027.599,E2 -2027.599} C_VEL
LIN {X 0,Y 573.227,Z 215.582,A -85,B 0,C 180,E1 -2030.391,E2 -2030.391} C_VEL
LIN {X 0,Y 573.311,Z 215.753,A -85,B 0,C 180,E1 -2031.377,E2 -2031.377} C_VEL
LIN {X 0,Y 573.621,Z 220.712,A -85,B 0,C 180,E1 -2032.222,E2 -2032.222} C_VEL
LIN {X 0,Y 573.468,Z 238.461,A -85,B 0,C 180,E1 -2035.186,E2 -2035.186} C_VEL
LIN {X 0,Y 573.308,Z 256.468,A -85,B 0,C 180,E1 -2038.15,E2 -2038.15} C_VEL
LIN {X 0,Y 573.443,Z 258.035,A -85,B 0,C 180,E1 -2038.239,E2 -2038.239} C_VEL
LIN {X 0,Y 574.084,Z 262.49,A -85,B 0,C 180,E1 -2038.314,E2 -2038.314} C_VEL
LIN {X 0,Y 573.866,Z 364.134,A -85,B 0,C 180,E1 -2039.606,E2 -2039.606} C_VEL
LIN {X 0,Y 573.784,Z 377.28,A -85,B 0,C 180,E1 -2039.917,E2 -2039.917} C_VEL
LIN {X 0,Y 573.702,Z 389.437,A -85,B 0,C 180,E1 -2040.342,E2 -2040.342} C_VEL
LIN {X 0,Y 573.605,Z 400.427,A -85,B 0,C 180,E1 -2040.854,E2 -2040.854} C_VEL
LIN {X 0,Y 573.47,Z 411.578,A -85,B 0,C 180,E1 -2041.519,E2 -2041.519} C_VEL
LIN {X 0,Y 573.338,Z 422.481,A -85,B 0,C 180,E1 -2042.337,E2 -2042.337} C_VEL
LIN {X 0,Y 573.25,Z 431.427,A -85,B 0,C 180,E1 -2043.162,E2 -2043.162} C_VEL
LIN {X 0,Y 573.155,Z 440.586,A -85,B 0,C 180,E1 -2044.196,E2 -2044.196} C_VEL
LIN {X 0,Y 573.064,Z 448.751,A -85,B 0,C 180,E1 -2045.356,E2 -2045.356} C_VEL
LIN {X 0,Y 573.03,Z 455.165,A -85,B 0,C 180,E1 -2046.509,E2 -2046.509} C_VEL
LIN {X 0,Y 572.969,Z 460.066,A -85,B 0,C 180,E1 -2047.651,E2 -2047.651} C_VEL
LIN {X 0,Y 572.968,Z 463.637,A -85,B 0,C 180,E1 -2048.767,E2 -2048.767} C_VEL
LIN {X 0,Y 572.968,Z 466.162,A -85,B 0,C 180,E1 -2049.913,E2 -2049.913} C_VEL
LIN {X 0,Y 572.963,Z 467.367,A -85,B 0,C 180,E1 -2050.802,E2 -2050.802} C_VEL
LIN {X 0,Y 572.933,Z 467.985,A -85,B 0,C 180,E1 -2052.141,E2 -2052.141} C_VEL
LIN {X 0,Y 572.978,Z 467.572,A -85,B 0,C 180,E1 -2053.063,E2 -2053.063} C_VEL
LIN {X 0,Y 572.95,Z 465.87,A -85,B 0,C 180,E1 -2054.344,E2 -2054.344} C_VEL
LIN {X 0,Y 572.991,Z 462.64,A -85,B 0,C 180,E1 -2055.667,E2 -2055.667} C_VEL
LIN {X 0,Y 573,Z 458.295,A -85,B 0,C 180,E1 -2056.885,E2 -2056.885} C_VEL
LIN {X 0,Y 573.042,Z 452.22,A -85,B 0,C 180,E1 -2058.145,E2 -2058.145} C_VEL
LIN {X 0,Y 573.113,Z 445.329,A -85,B 0,C 180,E1 -2059.253,E2 -2059.253} C_VEL
LIN {X 0,Y 573.195,Z 437.279,A -85,B 0,C 180,E1 -2060.294,E2 -2060.294} C_VEL
LIN {X 0,Y 573.265,Z 428.86,A -85,B 0,C 180,E1 -2061.185,E2 -2061.185} C_VEL
LIN {X 0,Y 573.395,Z 418.488,A -85,B 0,C 180,E1 -2062.074,E2 -2062.074} C_VEL
LIN {X 0,Y 573.499,Z 406.851,A -85,B 0,C 180,E1 -2062.872,E2 -2062.872} C_VEL
LIN {X 0,Y 573.636,Z 395.401,A -85,B 0,C 180,E1 -2063.487,E2 -2063.487} C_VEL
LIN {X 0,Y 573.743,Z 383.34,A -85,B 0,C 180,E1 -2063.979,E2 -2063.979} C_VEL
LIN {X 0,Y 573.829,Z 370.401,A -85,B 0,C 180,E1 -2064.355,E2 -2064.355} C_VEL
LIN {X 0,Y 573.89,Z 358.185,A -85,B 0,C 180,E1 -2064.576,E2 -2064.576} C_VEL
LIN {X 0,Y 573.955,Z 261.033,A -85,B 0,C 180,E1 -2065.798,E2 -2065.798} C_VEL
LIN {X 0,Y 573.329,Z 256.931,A -85,B 0,C 180,E1 -2065.892,E2 -2065.892} C_VEL
LIN {X 0,Y 573.38,Z 242.447,A -85,B 0,C 180,E1 -2068.244,E2 -2068.244} C_VEL
LIN {X 0,Y 573.571,Z 226.658,A -85,B 0,C 180,E1 -2070.877,E2 -2070.877} C_VEL
LIN {X 0,Y 573.575,Z 217.321,A -85,B 0,C 180,E1 -2072.458,E2 -2072.458} C_VEL
LIN {X 0,Y 573.284,Z 215.628,A -85,B 0,C 180,E1 -2072.81,E2 -2072.81} C_VEL
LIN {X 0,Y 573.29,Z 215.569,A -85,B 0,C 180,E1 -2075.628,E2 -2075.628} C_VEL
LIN {X 0,Y 573.287,Z 215.569,A -85,B 0,C 180,E1 -2077.75,E2 -2077.75} C_VEL
LIN {X 0,Y 573.264,Z 215.581,A -85,B 0,C 180,E1 -2080.596,E2 -2080.596} C_VEL
LIN {X 0,Y 573.232,Z 215.575,A -85,B 0,C 180,E1 -2083.47,E2 -2083.47} C_VEL
LIN {X 0,Y 573.251,Z 215.572,A -85,B 0,C 180,E1 -2085.647,E2 -2085.647} C_VEL
LIN {X 0,Y 573.226,Z 215.574,A -85,B 0,C 180,E1 -2087.849,E2 -2087.849} C_VEL
LIN {X 0,Y 573.24,Z 215.58,A -85,B 0,C 180,E1 -2090.826,E2 -2090.826} C_VEL
LIN {X 0,Y 573.26,Z 215.579,A -85,B 0,C 180,E1 -2093.164,E2 -2093.164} C_VEL
LIN {X 0,Y 573.254,Z 215.568,A -85,B 0,C 180,E1 -2096.19,E2 -2096.19} C_VEL
LIN {X 0,Y 573.233,Z 215.572,A -85,B 0,C 180,E1 -2098.564,E2 -2098.564} C_VEL
LIN {X 0,Y 573.225,Z 215.579,A -85,B 0,C 180,E1 -2100.993,E2 -2100.993} C_VEL
LIN {X 0,Y 573.266,Z 215.578,A -85,B 0,C 180,E1 -2103.534,E2 -2103.534} C_VEL
LIN {X 0,Y 573.255,Z 215.573,A -85,B 0,C 180,E1 -2106.048,E2 -2106.048} C_VEL
LIN {X 0,Y 573.225,Z 215.575,A -85,B 0,C 180,E1 -2108.702,E2 -2108.702} C_VEL
LIN {X 0,Y 573.227,Z 215.579,A -85,B 0,C 180,E1 -2111.457,E2 -2111.457} C_VEL
LIN {X 0,Y 573.234,Z 215.576,A -85,B 0,C 180,E1 -2114.333,E2 -2114.333} C_VEL
LIN {X 0,Y 573.226,Z 215.576,A -85,B 0,C 180,E1 -2116.647,E2 -2116.647} C_VEL
LIN {X 0,Y 573.24,Z 215.574,A -85,B 0,C 180,E1 -2119.481,E2 -2119.481} C_VEL
LIN {X 0,Y 573.213,Z 215.584,A -85,B 0,C 180,E1 -2122.197,E2 -2122.197} C_VEL
LIN {X 0,Y 573.26,Z 215.573,A -85,B 0,C 180,E1 -2124.822,E2 -2124.822} C_VEL
LIN {X 0,Y 573.235,Z 215.573,A -85,B 0,C 180,E1 -2127.359,E2 -2127.359} C_VEL
LIN {X 0,Y 573.235,Z 215.574,A -85,B 0,C 180,E1 -2129.828,E2 -2129.828} C_VEL
LIN {X 0,Y 573.27,Z 215.571,A -85,B 0,C 180,E1 -2132.239,E2 -2132.239} C_VEL
LIN {X 0,Y 573.25,Z 215.574,A -85,B 0,C 180,E1 -2135.125,E2 -2135.125} C_VEL
LIN {X 0,Y 573.242,Z 215.573,A -85,B 0,C 180,E1 -2137.667,E2 -2137.667} C_VEL
LIN {X 0,Y 573.265,Z 215.577,A -85,B 0,C 180,E1 -2140.731,E2 -2140.731} C_VEL
LIN {X 0,Y 573.247,Z 215.57,A -85,B 0,C 180,E1 -2143.626,E2 -2143.626} C_VEL
LIN {X 0,Y 573.262,Z 215.568,A -85,B 0,C 180,E1 -2145.811,E2 -2145.811} C_VEL
LIN {X 0,Y 573.274,Z 215.57,A -85,B 0,C 180,E1 -2148.738,E2 -2148.738} C_VEL
LIN {X 0,Y 573.3,Z 215.573,A -85,B 0,C 180,E1 -2151.544,E2 -2151.544} C_VEL
LIN {X 0,Y 573.289,Z 215.565,A -85,B 0,C 180,E1 -2154.375,E2 -2154.375} C_VEL
LIN {X 0,Y 573.305,Z 215.566,A -85,B 0,C 180,E1 -2157.896,E2 -2157.896} C_VEL
LIN {X 0,Y 573.329,Z 215.56,A -85,B 0,C 180,E1 -2160.705,E2 -2160.705} C_VEL
LIN {X 0,Y 573.306,Z 215.564,A -85,B 0,C 180,E1 -2162.814,E2 -2162.814} C_VEL
LIN {X 0,Y 573.285,Z 215.573,A -85,B 0,C 180,E1 -2165.631,E2 -2165.631} C_VEL
LIN {X 0,Y 573.283,Z 215.568,A -85,B 0,C 180,E1 -2168.462,E2 -2168.462} C_VEL
LIN {X 0,Y 573.273,Z 215.566,A -85,B 0,C 180,E1 -2171.315,E2 -2171.315} C_VEL
LIN {X 0,Y 573.283,Z 215.575,A -85,B 0,C 180,E1 -2174.426,E2 -2174.426} C_VEL
LIN {X 0,Y 573.262,Z 215.57,A -85,B 0,C 180,E1 -2177.114,E2 -2177.114} C_VEL
LIN {X 0,Y 573.245,Z 215.575,A -85,B 0,C 180,E1 -2180.079,E2 -2180.079} C_VEL
LIN {X 0,Y 573.236,Z 215.578,A -85,B 0,C 180,E1 -2182.34,E2 -2182.34} C_VEL
LIN {X 0,Y 573.247,Z 215.573,A -85,B 0,C 180,E1 -2185.413,E2 -2185.413} C_VEL
LIN {X 0,Y 573.239,Z 215.579,A -85,B 0,C 180,E1 -2188.567,E2 -2188.567} C_VEL
LIN {X 0,Y 573.224,Z 215.584,A -85,B 0,C 180,E1 -2190.996,E2 -2190.996} C_VEL
LIN {X 0,Y 573.247,Z 215.575,A -85,B 0,C 180,E1 -2193.522,E2 -2193.522} C_VEL
LIN {X 0,Y 573.198,Z 215.577,A -85,B 0,C 180,E1 -2196.055,E2 -2196.055} C_VEL
LIN {X 0,Y 573.243,Z 215.575,A -85,B 0,C 180,E1 -2198.703,E2 -2198.703} C_VEL
LIN {X 0,Y 573.233,Z 215.579,A -85,B 0,C 180,E1 -2201.594,E2 -2201.594} C_VEL
LIN {X 0,Y 573.227,Z 215.571,A -85,B 0,C 180,E1 -2204.336,E2 -2204.336} C_VEL
LIN {X 0,Y 573.241,Z 215.578,A -85,B 0,C 180,E1 -2207.36,E2 -2207.36} C_VEL
LIN {X 0,Y 573.241,Z 215.573,A -85,B 0,C 180,E1 -2210.393,E2 -2210.393} C_VEL
LIN {X 0,Y 573.236,Z 215.574,A -85,B 0,C 180,E1 -2213.077,E2 -2213.077} C_VEL
LIN {X 0,Y 573.268,Z 215.577,A -85,B 0,C 180,E1 -2215.672,E2 -2215.672} C_VEL
LIN {X 0,Y 573.242,Z 215.581,A -85,B 0,C 180,E1 -2218.185,E2 -2218.185} C_VEL
LIN {X 0,Y 573.247,Z 215.575,A -85,B 0,C 180,E1 -2220.634,E2 -2220.634} C_VEL
LIN {X 0,Y 573.225,Z 215.576,A -85,B 0,C 180,E1 -2223.023,E2 -2223.023} C_VEL
LIN {X 0,Y 573.24,Z 215.575,A -85,B 0,C 180,E1 -2225.365,E2 -2225.365} C_VEL
LIN {X 0,Y 573.292,Z 215.735,A -85,B 0,C 180,E1 -2227.665,E2 -2227.665} C_VEL
LIN {X 0,Y 573.855,Z 220.465,A -85,B 0,C 180,E1 -2228.444,E2 -2228.444} C_VEL
LIN {X 0,Y 573.666,Z 239.853,A -85,B 0,C 180,E1 -2231.426,E2 -2231.426} C_VEL
LIN {X 0,Y 573.43,Z 259.158,A -85,B 0,C 180,E1 -2234.358,E2 -2234.358} C_VEL
LIN {X 0,Y 573.371,Z 271.296,A -85,B 0,C 180,E1 -2236.149,E2 -2236.149} C_VEL
LIN {X 0,Y 574.077,Z 276.532,A -85,B 0,C 180,E1 -2236.257,E2 -2236.257} C_VEL
LIN {X 0,Y 573.884,Z 378.961,A -85,B 0,C 180,E1 -2237.558,E2 -2237.558} C_VEL
LIN {X 0,Y 573.794,Z 392.228,A -85,B 0,C 180,E1 -2237.87,E2 -2237.87} C_VEL
LIN {X 0,Y 573.679,Z 405.502,A -85,B 0,C 180,E1 -2238.339,E2 -2238.339} C_VEL
LIN {X 0,Y 573.591,Z 416.738,A -85,B 0,C 180,E1 -2238.88,E2 -2238.88} C_VEL
LIN {X 0,Y 573.432,Z 428.204,A -85,B 0,C 180,E1 -2239.585,E2 -2239.585} C_VEL
LIN {X 0,Y 573.328,Z 438.605,A -85,B 0,C 180,E1 -2240.386,E2 -2240.386} C_VEL
LIN {X 0,Y 573.238,Z 447.078,A -85,B 0,C 180,E1 -2241.185,E2 -2241.185} C_VEL
LIN {X 0,Y 573.161,Z 454.963,A -85,B 0,C 180,E1 -2242.071,E2 -2242.071} C_VEL
LIN {X 0,Y 573.076,Z 462.949,A -85,B 0,C 180,E1 -2243.185,E2 -2243.185} C_VEL
LIN {X 0,Y 573.07,Z 469.681,A -85,B 0,C 180,E1 -2244.37,E2 -2244.37} C_VEL
LIN {X 0,Y 573.029,Z 474.373,A -85,B 0,C 180,E1 -2245.428,E2 -2245.428} C_VEL
LIN {X 0,Y 573.022,Z 477.958,A -85,B 0,C 180,E1 -2246.484,E2 -2246.484} C_VEL
LIN {X 0,Y 572.959,Z 479.809,A -85,B 0,C 180,E1 -2247.188,E2 -2247.188} C_VEL
LIN {X 0,Y 572.946,Z 482.186,A -85,B 0,C 180,E1 -2248.594,E2 -2248.594} C_VEL
LIN {X 0,Y 572.938,Z 483,A -85,B 0,C 180,E1 -2250,E2 -2250} C_VEL
LIN {X 0,Y 572.946,Z 482.186,A -85,B 0,C 180,E1 -2251.406,E2 -2251.406} C_VEL
LIN {X 0,Y 572.938,Z 481.199,A -85,B 0,C 180,E1 -2252.109,E2 -2252.109} C_VEL
LIN {X 0,Y 572.959,Z 479.809,A -85,B 0,C 180,E1 -2252.813,E2 -2252.813} C_VEL
LIN {X 0,Y 573.015,Z 476.895,A -85,B 0,C 180,E1 -2253.868,E2 -2253.868} C_VEL
LIN {X 0,Y 572.963,Z 472.948,A -85,B 0,C 180,E1 -2254.926,E2 -2254.926} C_VEL
LIN {X 0,Y 573.068,Z 466.875,A -85,B 0,C 180,E1 -2256.16,E2 -2256.16} C_VEL
